"B_MA_SKZ_HydraulikEin"	MB 132	BYTE	// MA: Schrittkette Hydraulik Ein
"B_MA_SKZ_Schmierung"	MB 133	BYTE	// MA: Schrittkette Schmierung
"B_MA_SKZ_Schmierzyklus"	MB 134	BYTE	// MA: Schrittkette Schmierzyklus
"B_MA_Entprell_Zaehler"	MB 135	BYTE	// MA: Entprellzaehler Schmierzyklus
"MB_RDY_M180_189"	MB 144	BYTE	// M180_189: Rückmeldungen
"MB_LED_Zustand_Retten"	MB 151	BYTE
"LED_Zustand_Retten"	MB 154	BYTE	// LED Zustand  retten bei Baustein FC_BHG
"B_MAG_SKZ_Magazin"	MB 162	BYTE	// MAG: Schrittkettenzaehler Magazin
"MB_SKZ_FD_SCHMIERUNG"	MB 163	BYTE
"B_SKZ_Ablauf"	MB 172	BYTE	// WZW: SKZ Ablauf
"B_MAG_SKZ_Unterbrechung"	MB 174	BYTE	// MAG: Schrittkettenzaehler Magunterbrechung
"MB_Zähler_Satus"	MB 177	BYTE	// Zähler im Statusmodul PW
"B_Pos_Speicher"	MB 178	BYTE	// PW: Pos Speicher
"B_Pos_Speicher_Alt"	MB 184	BYTE	// PW: Pos Speicher Alt
"MB_Bruch1"	MB 185	BYTE	// PW: SKZ Fehlermodul
"MB_PW_Pos"	MB 188	BYTE	// SKZ Palettenträger drehen
"MB_WZSP_beide_As_1"	MB 192	BYTE	// WSP: Zaehler f. Verzoeg. beide Eingaenge 1 Signal
"MB_SKZ_PWAblauf"	MB 193	BYTE	// PW: SKZ Ablauf
"MB_WZSP_SKZ_Ablaufmodul"	MB 194	BYTE	// WSP: Schrittkettenzaehler Ablaufmodul Werkzeugspanner
"MB_Counter_Verzoe_Oeffn"	MB 196	BYTE	// WSP: Zaehler fuer verzoegertes oeffnen
"MB_Counter_Verzoe_NotAus"	MB 198	BYTE	// WSP: Zaehler fuer Verzoegerung nach Not-Aus und M6 Request
"MB_INIT_ASUP"	MB 200	BYTE	// ASUP:Initialisierung
"Start_ASUP_Machine"	MB 201	BYTE	// ASUP-fc201
"MB_START_ASUP`S"	MB 202	BYTE
"Start_ASUP_Frame"	MB 203	BYTE	// ASUP-fc203
"MB_A_ASpOV"	MB 204	BYTE
"MB_SKZ_Feierabend"	MB 211	BYTE	// PID: Schrittkettenzähler Feierabendschaltung
"B_SPos_Speicher"	MB 220	BYTE	// SCHWENKKOPF:Pos Speicher
"B_SPos_Speicher_Alt"	MB 221	BYTE	// SCHWENKKOPF:Pos Speicher Alt
"B_SKZ_SErr"	MB 222	BYTE	// SCHWENKKOPF:SKZ Fehlermodul
"B_SKZ_SStat"	MB 223	BYTE	// SCHWENKKOPF:SKZ Statusmodul
"B_SK_Ablauf"	MB 226	BYTE	// SCHWENKKOPF:SKZ Ablauf
"MB_aktiver_Verfahrbereic"	MB 228	BYTE
"MB_SKR_SKZ"	MB 230	BYTE	// SOFTKEYRETTUNG: Schrittkettenzaehler
"M_SPF_SKZ"	MB 242	BYTE	// SPF: Schrittkettenzaehler Spaenefoerderer
"MB_SPF_Zeit_Zaehler"	MB 243	BYTE	// SPF: Zähler für Spänefoerderer Zeiten
"MB_SKZ_RundachsAnf"	MB 247	BYTE	// AX: SKZ Anforderungen Rundachsmodul
"MB_5Achs_Typ"	MB 250	BYTE	// AX: Typ der 5 Achse
"MB_6Achs_Typ"	MB 251	BYTE	// AX: Typ der 10. Achse 6-te Seite
"MB_M10_11_Achse"	MB 256	BYTE	// AX: Zurordnung Achse M10/11
"MB_M22_23_Achse"	MB 257	BYTE	// AX: Zurordnung Achse M22/23
"MB_M32_33_Achse"	MB 258	BYTE	// AX: Zurordnung Achse M32/33
"MB_4Achs_Typ"	MB 259	BYTE	// AX: Typ der 4 Achse
"MB_4Achs_Konfig"	MB 262	BYTE	// AX: Konfiguration der 4. Achse
"MB_5Achs_Konfig"	MB 263	BYTE	// AX: Konfiguration der 5. Achse
"MB_6Achs_Konfig"	MB 264	BYTE	// AX: Konfiguration der 10. Achse 6-te Seite
"MB_SKZ_4ACHS"	MB 265	BYTE	// AX: Schrittkettenzaehler 4. Achse
"MB_SKZ_5ACHS"	MB 266	BYTE	// AX: Schrittkettenzaehler 5./11. Achse
"MB_SKZ_6ACHS"	MB 267	BYTE
"MB_FD_SCHM_HUEBE"	MB 271	BYTE
"MB_FD_ANZAHL_SCHMIERHUB"	MB 272	BYTE
"M_SKZ_Be_Entladen"	MB 292	BYTE	// WZW: SKZ Be-/Entladen
"B_SKZ_Reinig"	MB 294	BYTE	// WZW: Schrittkette Reinigen
"MB_Wiko_NCSNR_alt"	MB 305	BYTE
"B_LS_Pos_Speicher"	MB 311	BYTE
"B_LS_Pos_Speicher_Alt"	MB 312	BYTE
"B_SKZ_LS_Werr"	MB 313	BYTE
"MB_SKZ_Transport"	MB 314	BYTE
"MB_SKZ_Drehstation"	MB 323	BYTE
"MB_SKZ_VERTMAG_WZW"	MB 369	BYTE
"MB_I_DM_ACHSTASTEN"	MB 370	BYTE	// MB-EINGANG: MSST Achstasten 1
"MB_KMTL_DS1_Zahler"	MB 380	BYTE
"MB_KMTL_DS2_Zahler"	MB 381	BYTE
"MB_VS_Korr_BHG"	MB 395	BYTE
"MB_Eil_Korr_BHG"	MB 396	BYTE
"A_Status_FC_PROG_LOAD"	MB 406	BYTE	// A-Status-Meldung von Baustein FC_PROG_LOAD_UNLOAD
"A_Error_FC_PROG_LOAD"	MB 407	BYTE	// A-Error-Meldung von Baustein FC_PROG_LOAD_UNLOAD
"MB_SKZ_Hub_PS"	MB 412	BYTE
"MB_SPF_links_rechts"	MB 429	BYTE
"MB_A_SpOV"	MB 468	BYTE	// Spindeloverride
"MB_SKZ_Getriebe"	MB 469	BYTE	// Getriebe: Schrittkettenzaehler
"MB_Getr_AnzVersuch"	MB 470	BYTE	// Getriebe: Anzahl Versuche
"B_SKZ_SFKSchmieroel"	MB 471	BYTE	// SS: SKZ Schmieröl Spindel
"MB_Werkzeugbruch"	MB 500	BYTE
"MB_WZW_SKZ_Old"	MB 501	BYTE
"MB_AX11_Positionierung"	MB 502	BYTE
"MB_SKZ_NCTAchse"	MB 504	BYTE
"MB_NCTAchs_Typ"	MB 516	BYTE	// AX: Typ der 11. Achse (NC-Teilapperat)
"MB_NCTAchs_Konfig"	MB 517	BYTE	// AX: Konfiguration der 11. Achse (NC-Teilapperat)
"MB_Kegelreinigung_VM_SKZ"	MB 548	BYTE
"mb_hmi_pro_zeilennummer"	MB 554	BYTE	// HMI-PRO: Einrichtzeilennummer
"MB_Palnum_auf_Uebergabep"	MB 556	BYTE	// Palettennummer auf Übergabeplatz
"I_Direkttasten_links"	MB 588	BYTE	// HMI-PRO: OP12/OP15A Direkttasten links
"I_Direkttasten_rechts"	MB 589	BYTE	// HMI-PRO: OP12/OP15A Direkttasten rechts
"MB_ADRESS_BYTE_1_EROWA"	MB 602	BYTE	// Adress Byte 1 der EROWA Schnittstelle
"MB_ADRESS_BYTE_2_EROWA"	MB 603	BYTE	// Adress Byte 2 der EROWA Schnittstelle
"MB_RPC_MODE"	MB 629	BYTE
"MB_RPC_MODE_OLD"	MB 630	BYTE
"MB_ACCESS_LEVEL"	MB 707	BYTE
"IB_GEN_OM_BYTE"	MB 708	BYTE	// Merkereingangsbyte von Smartkey-Reader
"MB_SMARTKEY_BYTE_1"	MB 814	BYTE
"MB_SMARTKEY_AUTHOR"	MB 815	BYTE	// Einstellung des Smartkey Identifizierung
"MB_SF_Rechen1_Co_Vor"	MB 1090	BYTE	// Zähler Sollposition Rechen1 vor  nicht erreicht
"MB_SF_Rechen1_Co_Zurueck"	MB 1091	BYTE	// Zähler Sollposition Rechen1 zurück  nicht erreicht
"MB_SF_Rechen2_Co_Vor"	MB 1095	BYTE
"MB_SF_Rechen2_Co_Zurueck"	MB 1096	BYTE	// Zähler Sollposition Rechen2 zurück  nicht erreicht
"MB_Tisch_Zeit Klem"	MB 1097	BYTE	// Zeit  Druckerhoehung Tisch Achse 200Bar
"MB_Tisch_Takt"	MB 1098	BYTE	// Zähler Tisch geklemmt bei Drucherhoehung 200 Bar
"MB_PERIPHERIE_E_BYTE66"	MB 2066	BYTE	// Zwischenspeicher Peripherie-Eingangsbyte 66
"MB_PERIPHERIE_E_BYTE63"	MB 2067	BYTE	// Zwischenspeicher Peripherie-Eingangsbyte 63
"MB_PERIPHERIE_E_BYTE505"	MB 2068	BYTE	// Digitaleingabemodul , PROFIsafe V2 (PEB505 = DB18.DBB38)
"MB_PERIPHERIE_A_BYTE76"	MB 2076	BYTE	// Zwischenspeicher Peripherie-Ausgangsbyte 76
"MD_VIBS_Eing_SP"	MD 328	REAL	// Skalierte Eingangsspannung des Vibrationssensors
"MD_Restweg_Ax3"	MD 422	REAL
"MD_TDS_FC197"	MD 478	DWORD
"MD_SPI_SPEED_ABS"	MD 726	REAL	// Betragswert der aktuellen Ist-Spindeldrehzahl
"MD_MAPAL_PROFIL"	MD 2040	DWORD	// Angewähltes Profil der U-Achse Mapal
"MW_Wort_0"	MW 0	WORD
"MW_Wort_2"	MW 2	WORD
"MW_Wort_4"	MW 4	WORD
"SpTransp_holen_von"	MW 30	WORD
"SpTransp_bringen_zu"	MW 32	WORD
"MW_BHG_Vorschub"	MW 40	WORD
"MW_DrehDurch_Zaehler"	MW 62	WORD	// DrehDurchführung: Zaehler
"MW_Nr_Bereitst"	MW 64	INT	// WZV: Bereitstellungsplatznummer
"MW_Mag_Plaetze_verfahren"	MW 76	WORD	// GT MAG1: Anzahl verfahrene Paletze bei Ref. Punkt suchen
"MW_Max_ZaehlImpuls"	MW 78	WORD	// GT MAG1: Maximale Zeit Aenderung Zaehlimpuls
"MW_MAG_TMP_Anforderung"	MW 100	WORD	// WZV: T Befehl Platz Anforderung
"MW_MAG_TMMP_Anforderung"	MW 102	WORD	// WZV: TM Platz Anforderung
"MW_Wert_Vibrsensor"	MW 116	INT	// Wert von Vibrationssensor
"I_FD_PT100"	MW 118	WORD	// Temperatursensor Pt100 Fraes-Drehtisch
"W_CHAN1_Flanken"	MW 122	WORD	// Kanal1 Flanken
"MW_Anz_Achs_SA"	MW 128	INT	// Anzahl Achsen Sonderbetriebsart
"MW_MAG_MP_Anforderung"	MW 164	WORD	// MAG: Magazinplatz Anforderung
"MW_MAG_MP_Ist"	MW 166	WORD	// MAG: Magazinplatz Istwert
"MW_MAG_MP_Soll"	MW 168	WORD	// MAG: Magazinplatz Sollwert
"MW_4A_Zust_Stern_Dreieck"	MW 174	WORD
"MW_Zeit_Feierabend"	MW 212	WORD	// PID: Zeitzähler Feierabendschaltung
"MW_BHG"	MW 218	INT
"MW_SFunct1"	MW 274	WORD
"Z_MW_ZYkl_Kratzf."	MW 276	WORD	// KMTL: Zeitzähler Kratzförderer
"MW_Kuehl_Agg_Count"	MW 278	WORD
"MW_SKZ_PWAblauf"	MW 324	INT
"MW_TNUMMER_WZLISTE"	MW 325	INT
"MW_WMR_CNC_EMPF_STORE"	MW 348	INT
"MW_OW_WMR_CNC_SENDEN"	MW 350	WORD	// OW_WMR_CNC_SENDEN vom letzten PLC-Zyklus
"MW_PW_Anwahl_Typ"	MW 362	INT
"MW_PW_Anwahl_Option"	MW 364	INT
"MW_PW_Anwahl_Option2"	MW 366	INT
"O_KM_PROP_VENTIL2"	MW 398	INT	// Proportionalventil Kuehlmittel Hochdruckkreis 80bar
"MW_RET_VAL_SCALE"	MW 402	WORD
"MW_RPL_Bereich"	MW 408	INT
"MW_RPL_Position"	MW 410	INT
"MW_Zaehler_in_Bereich"	MW 415	WORD
"I_HCD1_MAL"	MW 422	INT	// MW-Eingang: Spannhydraulik Druckueberwachung Maschine
"I_HCD1_SST"	MW 424	INT	// MW-Eingang: Spannhydraulik Druckueberwachung Ruestplatz
"MW_SFunct"	MW 464	WORD	// S-Wert
"MW_Zust_Stern_Dreieck"	MW 466	WORD	// Stern Dreieck: Zustandszähler
"MW_SpiSchm_Zaehler"	MW 472	WORD	// Spindel-Schmierung Zähler
"MW_Mess_Nr"	MW 482	INT
"O_BIS_C_35"	MW 484	WORD	// Balluff
"MW_A_Position"	MW 486	WORD
"I_BIS_C_35"	MW 488	WORD	// MW-EINGÄNGE:
"MW_STATE_AXPOSLESEN"	MW 490	WORD
"O_BIS_C_35_1"	MW 492	WORD
"MW_SHOPM_Werkzeugkennung"	MW 494	WORD
"ErrCode_FC_SIEM_PLC_NCK"	MW 496	INT	// ErrCode von Baustein FC_SIEM_PLC_NCK
"WZV_T-Daten"	MW 498	WORD	// WZV: T-Daten neu lesen
"MW_Status_TM_TRANS"	MW 502	WORD
"O_BIS_C_35_2"	MW 504	WORD
"M_WZV_Gr2_WST"	MW 508	WORD	// WZV Zwischenspeicher asynchron Ablegen im Magazin
"MW_ERROR_TM_TRANS"	MW 510	WORD
"I_SPI_TEMP_LAG_HINTEN"	MW 512	WORD	// MW-EINGÄNGE:
"I_Temp_Analog_2"	MW 514	WORD	// MW-EINGÄNGE:
"O_KM_PROP_VENTIL1"	MW 518	INT	// MW-AUSGANG: Kühlmittel Hochdruck PROP-Ventil
"MW_Num_Chanels"	MW 542	WORD
"MW_WFK_NC_SNR"	MW 544	INT
"MW_WK_Nummer"	MW 546	INT
"O_VMS_SPI_SPEED_RPM"	MW 558	WORD
"MW_Greifer_ausfahren_SKZ"	MW 562	INT
"MW_numMagPlaceParam"	MW 570	INT	// Anzahl PArameter Magazinplaetze
"MW_Kegelreinigung_VM_SKZ"	MW 586	INT
"MW_SPF_Zeit_Zaehler"	MW 592	WORD
"MW_WERKSTUECK_ADRESSE"	MW 604	WORD	// Handlingsystem Werkstück Adresse aus H-Fkt 65 bzw. PAR2 in DM_M65
"MW_SERIELLE_ADRESSE"	MW 606	WORD	// Handlingsystem Serielle Adresse Komplett
"MW_ADRESSE_KONTR"	MW 610	WORD
"MW_VMS_SPI_SPEED_RPM"	MW 612	INT	// Analogausgang Vibrationssensor Spindeldrehzahl
"MW_VMS_VIBRATION_SPINDLE"	MW 616	INT	// Analogeingang Vibrationssensor Schwinggeschwindigkeit veff
"MW_RET_VAL_UNSCALE"	MW 618	WORD
"MW_STATUS_MASCH"	MW 624	WORD
"MW_STATUSMASCH_OLD"	MW 626	WORD
"MW_Teilung_RPL"	MW 650	INT
"MW_Teilung_RPL_alt"	MW 652	INT
"I_MACH_BED_T_COMP"	MW 664	WORD
"I_SPI_TEMP_BEA_FRONT"	MW 666	WORD
"I_VMS_VIBRATION_SPINDLE"	MW 668	WORD
"I_TUNING_CPU_KSA_0"	MW 674	WORD
"I_TUNING_CPU_KSA_1"	MW 676	WORD
"I_TUNING_CPU_KSA_2"	MW 678	WORD
"I_TUNING_CPU_KSA_3"	MW 680	WORD
"I_TUNING_CPU_KSA_4"	MW 682	WORD
"O_TUNING_CPU_KSA_0"	MW 684	WORD
"O_TUNING_CPU_KSA_1"	MW 686	WORD
"O_TUNING_CPU_KSA_2"	MW 688	WORD
"O_TUNING_CPU_KSA_3"	MW 690	WORD
"O_TUNING_CPU_KSA_4"	MW 692	WORD
"I_SPI_WZ_SPA"	MW 700	WORD	// Analoger Werkzeugspanner der Spindel
"I_SPI_VERLAG_SENSOR"	MW 702	WORD	// Axiale Wellenverlagerung Startwert Uzo GMN Spindel
"I_ML_SPI_1"	MW 710	WORD	// Merkerwort Eingang  MMS-Vogel
"O_ML_SPI_1"	MW 712	WORD	// Merkerwort Ausgang MMS-Vogel
"MW_SPI_REF_Zeitintervall"	MW 730	WORD	// Spindelüberwachung: Zeitintervall für Spindel Referenzlauf
"MW_PW_TIME_senken"	MW 736	INT	// Time Hub senken  bis PW in Mittelstellung
"MW_PW_Time_ausbl_kon"	MW 738	INT	// Zeitvorgabe Spuel-Konenluftleitung ausblasen
"MW_PW_Time_Spuel_resu"	MW 740	INT	// Resultierende Spuelzeit beim PW senken
"MW_PW_Time_spuel_senk"	MW 742	S5TIME	// Spuelzeit PW-Hub senken ohne Positionsschalter4
"MW_PW_Time_Zeitr_ausbl"	MW 744	S5TIME	// Timer ausblasen Konen
"MW_GetTNR_State"	MW 862	WORD	// State von Call GET_TNR
"MW_Get_Toolstate_State"	MW 864	WORD
"MW1_Get_Toolstate_State"	MW 866	WORD
"I_GEN_POWERMEAS_SPI"	MW 1086	WORD	// MW-Eingänge: Analogeingang Messung Leistung Hauptantrieb
"I_GEN_FLC_COOL_AG_2"	MW 1088	WORD	// MW-Eingänge: Messeinrichtung Kuehlmittel 2
"I_SPI_TEMP_LAG_VORNE"	MW 1092	WORD
"State_FB_SIEM_PUT_GUDs"	MW 1100	WORD	// State-meldung von Baustein FB_SIEM_PUT beim Ablegen der GUDs
"I_SPI_KABEL_PT100_1"	MW 1102	WORD	// MW-EINGÄNGE: Temperatursensor 1 Leitungsueberwachung Hauptantrieb
"I_SPI_KABEL_PT100_2"	MW 1104	WORD	// MW-EINGÄNGE: Temperatursensor 2 Leitungsueberwachung Hauptantrieb
"I_SPI_TEMP"	MW 1106	WORD
"I_MASCH_BETT_T_KOMP"	MW 1120	WORD	// MW-EINGÄNGE: Temperatursensor Maschinenbett PT 100
"I_SPI_PT100"	MW 1122	WORD	// MW-EINGÄNGE: Lager-Temperatursensor PT100 Hauptantrieb
"I_VSP_TEMP"	MW 1124	WORD
"I_SPI_TEMP_MONITOR"	MW 2000	WORD	// MW-EINGÄNGE: Temperaturüberwachung Spindelstock (55/65H)
"I_RESERVE_4_33"	MW 2002	WORD	// MW-EINGÄNGE: Dummy für Hardware 55H
"OB_ZYKLISCH"	OB 1	OB 1	// Zyklische Programmbearbeitung
"TOD_INT0"	OB 10	OB 10	// Time of Day Interrupt 0
"OB_WECKALARM1"	OB 35	OB 35	// Cyclic Interrupt 1
"OB_PROZESSALARM1"	OB 40	OB 40	// Prozessalarm 1
"OB_I_O_FLT1"	OB 82	OB 82	// I/O Point Fault 1
"OB_PRG_ABL_FEHLER"	OB 85	OB 85	// OB Programmablauffehler
"OB_RACK_FLT"	OB 86	OB 86	// Loss of Rack Fault
"OB_WARMSTART1"	OB 100	OB 100	// Hochlauf / Neustart
"OB_PROG_ERR"	OB 121	OB 121	// Programming Error
"OB_MOD_ERR"	OB 122	OB 122	// Module Access Error
"IB_HCD_AV_CL_PO_1_SST_H"	PIB 430	BYTE
"IB_HCD_AV_CL_PO_1_SST_L"	PIB 431	BYTE
"IB_HCD_AV_CL_PO_2_SST_H"	PIB 432	BYTE
"IB_HCD_AV_CL_PO_2_SST_L"	PIB 433	BYTE
"IB_HCD_AV_CL_PO_3_SST_H"	PIB 434	BYTE
"IB_HCD_AV_CL_PO_3_SST_L"	PIB 435	BYTE
"IB_HCD_AV_CL_PO_4_SST_H"	PIB 436	BYTE
"IB_HCD_AV_CL_PO_4_SST_L"	PIB 437	BYTE
"IB_HCD_AV_CL_PO_1_MPL_H"	PIB 438	BYTE
"IB_HCD_AV_CL_PO_1_MPL_L"	PIB 439	BYTE
"IB_HCD_AV_CL_PO_2_MPL_H"	PIB 440	BYTE
"IB_HCD_AV_CL_PO_2_MPL_L"	PIB 441	BYTE
"IB_HCD_AV_CL_PO_3_MPL_H"	PIB 442	BYTE
"IB_HCD_AV_CL_PO_3_MPL_L"	PIB 443	BYTE
"IB_HCD_AV_CL_PO_4_MPL_H"	PIB 444	BYTE
"IB_HCD_AV_CL_PO_4_MPL_L"	PIB 445	BYTE
"IB_HCD_STATE_CL_PO_1_SST"	PIB 446	BYTE
"IB_HCD_STATE_CL_PO_2_SST"	PIB 447	BYTE
"IB_HCD_STATE_CL_PO_3_SST"	PIB 448	BYTE
"IB_HCD_STATE_CL_PO_4_SST"	PIB 449	BYTE
"IB_HCD_STATE_CL_PO_1_MPL"	PIB 450	BYTE
"IB_HCD_STATE_CL_PO_2_MPL"	PIB 451	BYTE
"IB_HCD_STATE_CL_PO_3_MPL"	PIB 452	BYTE
"IB_HCD_STATE_CL_PO_4_MPL"	PIB 453	BYTE
"IB_HCD_DIAG_SOFTWARE"	PIB 454	BYTE
"IB_HCD_DIAG_MPL_SST"	PIB 455	BYTE
"IB_HCD_MI_TURNT_INP"	PIB 456	BYTE
"IB_SP_P_IST_ST_1_RPL_H"	PIB 1000	BYTE	// HAWE-Box:
"IB_SP_P_IST_ST_1_RPL_L"	PIB 1001	BYTE	// HAWE-Box:
"IB_SP_P_IST_ST_2_RPL_H"	PIB 1002	BYTE	// HAWE-Box:
"IB_SP_P_IST_ST_2_RPL_L"	PIB 1003	BYTE	// HAWE-Box:
"IB_SP_P_IST_ST_3_RPL_H"	PIB 1004	BYTE	// HAWE-Box:
"IB_SP_P_IST_ST_3_RPL_L"	PIB 1005	BYTE	// HAWE-Box:
"IB_SP_P_IST_ST_4_RPL_H"	PIB 1006	BYTE	// HAWE-Box:
"IB_SP_P_IST_ST_4_RPL_L"	PIB 1007	BYTE	// HAWE-Box:
"IB_SP_P_IST_ST_1_MPL_H"	PIB 1008	BYTE	// HAWE-Box:
"IB_SP_P_IST_ST_1_MPL_L"	PIB 1009	BYTE	// HAWE-Box:
"IB_SP_P_IST_ST_2_MPL_H"	PIB 1010	BYTE	// HAWE-Box:
"IB_SP_P_IST_ST_2_MPL_L"	PIB 1011	BYTE	// HAWE-Box:
"IB_SP_P_IST_ST_3_MPL_H"	PIB 1012	BYTE	// HAWE-Box:
"IB_SP_P_IST_ST_3_MPL_L"	PIB 1013	BYTE	// HAWE-Box:
"IB_SP_P_IST_ST_4_MPL_H"	PIB 1014	BYTE	// HAWE-Box:
"IB_SP_P_IST_ST_4_MPL_L"	PIB 1015	BYTE	// HAWE-Box:
"IB_SP_STATE_ST_1_RPL"	PIB 1016	BYTE	// HAWE-Box:
"IB_SP_STATE_ST_2_RPL"	PIB 1017	BYTE	// HAWE-Box:
"IB_SP_STATE_ST_3_RPL"	PIB 1018	BYTE	// HAWE-Box:
"IB_SP_STATE_ST_4_RPL"	PIB 1019	BYTE	// HAWE-Box:
"IB_SP_STATE_ST_1_MPL"	PIB 1020	BYTE	// HAWE-Box:
"IB_SP_STATE_ST_2_MPL"	PIB 1021	BYTE	// HAWE-Box:
"IB_SP_STATE_ST_3_MPL"	PIB 1022	BYTE	// HAWE-Box:
"IB_SP_STATE_ST_4_MPL"	PIB 1023	BYTE	// HAWE-Box:
"IB_SP_FUNKTION_MPL_RPL"	PIB 1024	BYTE	// HAWE-Box:
"IB_SP_DIAGNOSE_MPL_RPL"	PIB 1025	BYTE	// HAWE-Box:
"IB_TOOL_CUT_FORCE_1_MON"	PIB 1300	BYTE	// ARTIS/Toolinspect Eingangs-Byte 1
"IW_Tuning_CPU_0"	PIW 210	WORD	// xx-xx.x ME Datenschnittstelle Profibus(8)
"IW_Tuning_CPU_1"	PIW 212	WORD	// xx-xx.x ME Datenschnittstelle Profibus(8)
"IW_Tuning_CPU_2"	PIW 214	WORD	// xx-xx.x ME Datenschnittstelle Profibus(8)
"IW_Tuning_CPU_3"	PIW 216	WORD	// xx-xx.x ME Datenschnittstelle Profibus(8)
"IW_Tuning_CPU_4"	PIW 218	WORD	// xx-xx.x ME Datenschnittstelle Profibus(8)
"IW_TUNING_CPU_5"	PIW 220	WORD	// xx-xx.x ME Datenschnittstelle Profibus(8)
"IW_WMR_CNC_0"	PIW 258	WORD	// REGAL EXTERN Bit-Orientiertes Eingangswort 0
"IW_WMR_CNC_1"	PIW 260	WORD	// REGAL EXTERN Bit-Orientiertes Eingangswort 1
"IW_WMR_CNC_MAINCOMMAND"	PIW 262	WORD	// REGAL EXTERN Hauptkommando Nutzdaten
"IW_WMR_CNC_SUBCOMMAND"	PIW 264	WORD	// REGAL EXTERN Unterkommando Nutzdaten
"IW_WMR_CNC_1_DATA"	PIW 266	WORD	// REGAL EXTERN Kennung Nutzdaten 1 Wort
"IW_WMR_CNC_2_DATA"	PIW 268	WORD	// REGAL EXTERN Kennung Nutzdaten 2 Wort
"IW_WMR_CNC_SENDEN"	PIW 270	WORD	// REGAL EXTERN Handshake senden Zaehler
"IW_WMR_CNC_EMPFANGEN"	PIW 272	WORD	// REGAL EXTERN Handshake empfangen Zaehler
"IW_TUNING_CPU_CU_0"	PIW 300	WORD
"IW_TUNING_CPU_CU_1"	PIW 302	WORD
"IW_TUNING_CPU_CU_2"	PIW 304	WORD
"IW_TUNING_CPU_CU_3"	PIW 306	WORD
"IW_TUNING_CPU_CU_4"	PIW 308	WORD
"IW_SP_Wort_24"	PIW 334	WORD	// SpannHydraulik Wort 24
"IW_BIS_C_35"	PIW 1060	WORD
"IW_ROBOT_0"	PIW 1160	WORD	// xx-xx.x ME Start-Adr: Roboter-Schnittstelle - DPDP-Koppler
"OB_HCD_SV_CL_PO_1_SST_H"	PQB 430	BYTE
"OB_HCD_SV_CL_PO_1_SST_L"	PQB 431	BYTE
"OB_HCD_SV_CL_PO_2_SST_H"	PQB 432	BYTE
"OB_HCD_SV_CL_PO_2_SST_L"	PQB 433	BYTE
"OB_HCD_SV_CL_PO_3_SST_H"	PQB 434	BYTE
"OB_HCD_SV_CL_PO_3_SST_L"	PQB 435	BYTE
"OB_HCD_SV_CL_PO_4_SST_H"	PQB 436	BYTE
"OB_HCD_SV_CL_PO_4_SST_L"	PQB 437	BYTE
"OB_HCD_SV_CL_PO_1_MPL_H"	PQB 438	BYTE
"OB_HCD_SV_CL_PO_1_MPL_L"	PQB 439	BYTE
"OB_HCD_SV_CL_PO_2_MPL_H"	PQB 440	BYTE
"OB_HCD_SV_CL_PO_2_MPL_L"	PQB 441	BYTE
"OB_HCD_SV_CL_PO_3_MPL_H"	PQB 442	BYTE
"OB_HCD_SV_CL_PO_3_MPL_L"	PQB 443	BYTE
"OB_HCD_SV_CL_PO_4_MPL_H"	PQB 444	BYTE
"OB_HCD_SV_CL_PO_4_MPL_L"	PQB 445	BYTE
"OB_HCD_STATE_CL_PO_1_SST"	PQB 446	BYTE
"OB_HCD_STATE_CL_PO_2_SST"	PQB 447	BYTE
"OB_HCD_STATE_CL_PO_3_SST"	PQB 448	BYTE
"OB_HCD_STATE_CL_PO_4_SST"	PQB 449	BYTE
"OB_HCD_STATE_CL_PO_1_MPL"	PQB 450	BYTE
"OB_HCD_STATE_CL_PO_2_MPL"	PQB 451	BYTE
"OB_HCD_STATE_CL_PO_3_MPL"	PQB 452	BYTE
"OB_HCD_STATE_CL_PO_4_MPL"	PQB 453	BYTE
"OB_HCD_FCT_MPL_SST"	PQB 454	BYTE
"OB_HCD_DIAG_MPL_SST"	PQB 455	BYTE
"OB_HCD_TOL_VAL_PRE_REA"	PQB 456	BYTE
"OB_HCD_TOL_VAL_READJUST"	PQB 457	BYTE
"OB_HCD_TOL_VAL_EMSTP"	PQB 458	BYTE
"OB_HCD_DELTA_CONTROL"	PQB 459	BYTE
"OB_HCD_DELTA_REGULATION"	PQB 460	BYTE
"OB_HCD_PRESSURE_RELEASE"	PQB 461	BYTE
"OB_HCD_PRE_RET_VALV_OPEN"	PQB 462	BYTE
"OB_HCD_TIME_DELAY_CLAMP"	PQB 463	BYTE
"OB_HCD_RT_RET_VAL_OPEN"	PQB 464	BYTE
"OB_SP_P_SOLL_ST_1_RPL_H"	PQB 1000	BYTE	// HAWE-Box:
"OB_SP_P_SOLL_ST_1_RPL_L"	PQB 1001	BYTE	// HAWE-Box:
"OB_SP_P_SOLL_ST_2_RPL_H"	PQB 1002	BYTE	// HAWE-Box:
"OB_SP_P_SOLL_ST_2_RPL_L"	PQB 1003	BYTE	// HAWE-Box:
"OB_SP_P_SOLL_ST_3_RPL_H"	PQB 1004	BYTE	// HAWE-Box:
"OB_SP_P_SOLL_ST_3_RPL_L"	PQB 1005	BYTE	// HAWE-Box:
"OB_SP_P_SOLL_ST_4_RPL_H"	PQB 1006	BYTE	// HAWE-Box:
"OB_SP_P_SOLL_ST_4_RPL_L"	PQB 1007	BYTE	// HAWE-Box:
"OB_SP_P_SOLL_ST_1_MPL_H"	PQB 1008	BYTE	// HAWE-Box:
"OB_SP_P_SOLL_ST_1_MPL_L"	PQB 1009	BYTE	// HAWE-Box:
"OB_SP_P_SOLL_ST_2_MPL_H"	PQB 1010	BYTE	// HAWE-Box:
"OB_SP_P_SOLL_ST_2_MPL_L"	PQB 1011	BYTE	// HAWE-Box:
"OB_SP_P_SOLL_ST_3_MPL_H"	PQB 1012	BYTE	// HAWE-Box:
"OB_SP_P_SOLL_ST_3_MPL_L"	PQB 1013	BYTE	// HAWE-Box:
"OB_SP_P_SOLL_ST_4_MPL_H"	PQB 1014	BYTE	// HAWE-Box:
"OB_SP_P_SOLL_ST_4_MPL_L"	PQB 1015	BYTE	// HAWE-Box:
"OB_SP_STATE_ST_1_RPL"	PQB 1016	BYTE	// HAWE-Box:
"OB_SP_STATE_ST_2_RPL"	PQB 1017	BYTE	// HAWE-Box:
"OB_SP_STATE_ST_3_RPL"	PQB 1018	BYTE	// HAWE-Box:
"OB_SP_STATE_ST_4_RPL"	PQB 1019	BYTE	// HAWE-Box:
"OB_SP_STATE_ST_1_MPL"	PQB 1020	BYTE	// HAWE-Box:
"OB_SP_STATE_ST_2_MPL"	PQB 1021	BYTE	// HAWE-Box:
"OB_SP_STATE_ST_3_MPL"	PQB 1022	BYTE	// HAWE-Box:
"OB_SP_STATE_ST_4_MPL"	PQB 1023	BYTE	// HAWE-Box:
"OB_SP_FUNKTION_MPL_RPL"	PQB 1024	BYTE	// HAWE-Box:
"OB_SP_DIAGNOSE_MPL_RPL"	PQB 1025	BYTE	// HAWE-Box:
"OB_SP_P_TOL_DRUCK_ERREIC"	PQB 1026	BYTE	// HAWE-Box:
"OB_SP_P_TOL_NACHREGELN"	PQB 1027	BYTE	// HAWE-Box:
"OB_SP_P_TOL_NOTAUS"	PQB 1028	BYTE	// HAWE-Box:
"OB_SP_DELTA_STEUERUNG"	PQB 1029	BYTE	// HAWE-Box:
"OB_SP_DELTA_REGELUNG"	PQB 1030	BYTE	// HAWE-Box:
"OB_SP_P_LOESEDRUCK"	PQB 1031	BYTE	// HAWE-Box:
"OB_SP_P_DRUCK_RV_OEFFNEN"	PQB 1032	BYTE	// HAWE-Box:
"OB_SP_T_VERZ_SPANNEN"	PQB 1033	BYTE	// HAWE-Box:
"OB_SP_T_RV_OEFFNEN"	PQB 1034	BYTE	// HAWE-Box:
"OB_TOOL_CUT_FORCE_1_MON"	PQB 1300	BYTE	// ARTIS/Toolinspect Ausgangs-Byte 1
"OB_TOOL_CUT_FORCE_2_MON"	PQB 1301	BYTE	// ARTIS/Toolinspect Ausgangs-Byte 2
"OW_Tuning_CPU_0"	PQW 210	WORD	// xx-xx.x MA Datenschnittstelle Profibus(8)
"OW_Tuning_CPU_1"	PQW 212	WORD	// xx-xx.x MA Datenschnittstelle Profibus(8)
"OW_Tuning_CPU_2"	PQW 214	WORD	// xx-xx.x MA Datenschnittstelle Profibus(8)
"OW_Tuning_CPU_3"	PQW 216	WORD	// xx-xx.x MA Datenschnittstelle Profibus(8)
"OW_Tuning_CPU_4"	PQW 218	WORD	// xx-xx.x MA Datenschnittstelle Profibus(8)
"OW_Tuning_CPU_C0"	PQW 220	WORD	// xx-xx.x MA Datenschnittstelle Profibus(8)
"OW_Tuning_CPU_C1"	PQW 222	WORD	// xx-xx.x MA Datenschnittstelle Profibus(8)
"OW_Tuning_CPU_C2"	PQW 224	WORD	// xx-xx.x MA Datenschnittstelle Profibus(8)
"OW_Tuning_CPU_C3"	PQW 226	WORD	// xx-xx.x MA Datenschnittstelle Profibus(8)
"OW_Tuning_CPU_5"	PQW 228	WORD	// xx-xx.x MA Datenschnittstelle Profibus(8)
"OW_Tuning_CPU_6"	PQW 230	WORD	// xx-xx.x MA Datenschnittstelle Profibus(8)
"OW_TUNING_CPU_7"	PQW 232	WORD	// xx-xx.x MA Datenschnittstelle Profibus(8)
"OW_TUNING_CPU_8"	PQW 234	WORD
"OW_WMR_CNC_0"	PQW 258	WORD	// REGAL EXTERN Bit-Orientiertes Ausgangswort 0
"OW_WMR_CNC_1"	PQW 260	WORD	// REGAL EXTERN Bit-Orientiertes Ausgangswort 1
"OW_WMR_CNC_MAINCOMMAND"	PQW 262	WORD	// REGAL EXTERN Hauptkommando Nutzdaten
"OW_WMR_CNC_SUBCOMMAND"	PQW 264	WORD	// REGAL EXTERN Unterkommando Nutzdaten
"OW_WMR_CNC_1_DATA"	PQW 266	WORD	// REGAL EXTERN Kennung Nutzdaten 1 Wort
"OW_WMR_CNC_2_DATA"	PQW 268	WORD	// REGAL EXTERN Kennung Nutzdaten 2 Wort
"OW_WMR_CNC_SENDEN"	PQW 270	WORD	// REGAL EXTERN Handshake senden Zaehler
"OW_WMR_CNC_EMPFANGEN"	PQW 272	WORD	// REGAL EXTERN Handshake empfangen Zaehler
"OW_TUNING_CPU_CU_0"	PQW 300	WORD
"OW_TUNING_CPU_CU_1"	PQW 302	WORD
"OW_TUNING_CPU_CU_2"	PQW 304	WORD
"OW_TUNING_CPU_CU_3"	PQW 306	WORD
"OW_TUNING_CPU_CU_4"	PQW 308	WORD
"OW_TUNING_CPU_CU_5"	PQW 310	WORD
"OW_BIS_C_35"	PQW 1060	WORD	// Balluff
"OW_BIS_C_35_1"	PQW 1062	WORD
"OW_BIS_C_35_2"	PQW 1064	WORD
"OW_ROBOT_0"	PQW 1160	WORD	// xx-xx.x MA Start-Adr: Roboter-Schnittstelle - DPDP-Koppler
"MSSTLED BA AUTO"	Q 0.0	BOOL	// MSST: LED Betriebsart AUTO_LED 21
"DM_LED Spindel links"	Q 0.4	BOOL	// MSST: LED Spindel links_LED 10
"DM_LED Spindel Halt *"	Q 0.5	BOOL	// MSST: LED Spindel Halt *_LED 9
"DM_LED Spindel rechts"	Q 0.6	BOOL	// MSST: LED Spindel rechts_LED 8
"DM_LED Y-Achse plus"	Q 1.4	BOOL	// MSST: LED Y-Achse minus_LED 20
"DM_LED Z-Achse plus(3)"	Q 1.5	BOOL	// MSST: LED Z-Achse plus LED 19
"DM_LED 4-Achse rechts"	Q 1.6	BOOL	// MSST: LED 4-Achse (4)_rechts LED 38
"MSSTLED 1 INC"	Q 2.0	BOOL	// MSST: LED 1 INC_LED 14
"MSSTLED 10 INC"	Q 2.1	BOOL	// MSST: LED 10 INC_LED 24
"MSSTLED 100 INC"	Q 2.2	BOOL	// MSST: LED 100 INC_LED 34
"MSSTLED 1000 INC"	Q 2.3	BOOL	// MSST: LED 1000 INC_LED 44
"MSSTLED var. INC"	Q 2.5	BOOL	// MSST: LED var. INC_LED 4
"DM_LED 5/6Achsanwahl"	Q 4.5	BOOL	// MSST: LED Anwahl 5/6Achse
"DM_LED 5/6-Achse minus"	Q 4.6	BOOL	// MSST: LED 5/6-Achse minus LED 48
"DM_LED 5/6-Achse plus"	Q 4.7	BOOL	// MSST: LED 5/6-Achse plus LED 48
"DM_LED X-Achse minus(1)"	Q 5.0	BOOL	// MSST: LED X-Achse (1) minus LED 28
"DM_LED Eilgang"	Q 5.1	BOOL	// MSST: LED_Eilgang LED 29
"DM_LED X-Achse plus(1)"	Q 5.2	BOOL	// MSST: LED X-Achse (1) plus LED 30
"DM_LED Y-Achse minus"	Q 5.3	BOOL	// MSST: LED Y-Achse plus_LED 38
"DM_LED Z-Achse minus(3)"	Q 5.4	BOOL	// MSST: LED Z. Achse (3)minus_LED 39
"MSSTLED C-Achse (6)"	Q 5.5	BOOL	// MSST: LED C-Achse (6)_LED 40
"DM_LED_MKS_WKS"	Q 6.1	BOOL	// MSST: LED MKS_WKS
"DM_LED SpiOver_erhoeh"	Q 6.4	BOOL	// MSST: LED Spinbdeloverride erhoehen
"DM_LED_SpiOver_100%"	Q 6.5	BOOL	// MSST: LED Spindeloverride 100%
"DM_LED_SpiOver_reduz"	Q 6.6	BOOL	// MSST: LED Spindeloverride reduzieren
"DM_LED IKZ_ein_aus"	Q 7.0	BOOL	// MSST: LED IKZ EIN/AUS
"DM_LED Kühlmittel"	Q 7.1	BOOL	// MSST: LED Kühlmittel EIN/AUS
"DM_LED_WZSpanner"	Q 7.4	BOOL	// MSST: LED Werkzeugspanner auf zu
"OX_AL_XACHS_Bremse_auf"	Q 32.0	BOOL	// Ansteuerung Motorbremse X-Achse
"OX_AL_YACHS_Bremse_auf"	Q 32.1	BOOL	// Ansteuerung Motorbremse Y-Achse
"OX_AL_ZACHS_Bremse_auf"	Q 33.0	BOOL	// Ansteuerung Motorbremse Z-Achse
"OX_AL_4ACHS_Bremse_auf"	Q 33.1	BOOL	// Ansteuerung Motorbremse 4-Achse
"OX_AL_5ACHS_Bremse_auf"	Q 34.0	BOOL	// Ansteuerung Motorbremse 5-Achse
"OX_PW_ACHS_Bremse_auf"	Q 34.1	BOOL	// Achse 8 (PW)  Bremse lüften
"OX_SPI_WYE"	Q 35.0	BOOL	// Stern Dreieck: Ausgang Stern
"OX_SPI_DELTA"	Q 35.1	BOOL	// Stern Dreieck: Ausgang Dreieck
"OX_GEN_PLC_RDY"	Q 36.0	BOOL	// Maschine 'Ein'  (CNC PLC Betriebsbereit)
"OX_WM_Freigabe_re_li"	Q 36.1	BOOL	// Freigabe Werkzeugmagazin
"OX_PC_DOOR_UNLOCK"	Q 36.2	BOOL	// Magnetverriegelung Ruestplatz Palettenwechsler entriegeln
"OX_OMS_ON"	Q 36.3	BOOL	// Nebel- u.Rauchabscheider 'Ein'
"OX_PC_MPL_PALLET_RELEASE"	Q 37.0	BOOL	// Palette auf Tisch lösen
"OX_PC_MPL_PALLET_CLAMP"	Q 37.1	BOOL	// Palette auf Tisch spannen
"OX_SH_CLAMP_CLAMP"	Q 37.2	BOOL	// Schwenkfraeskopf Klemmung klemmen
"OX_SH_CLAMP_RELEASE"	Q 37.3	BOOL	// Schwenkfraeskopf Klemmung loesen
"OX_GEN_AXIS4_CLAMP"	Q 38.0	BOOL	// 4.Achse klemmen
"OX_GEN_AXIS5_CLAMP"	Q 38.1	BOOL	// 5.Achse klemmen
"OX_SPI_LUB_OIL_PUMP_ON"	Q 38.2	BOOL	// Schmierung Hauptantrieb 24.000 U/min
"OX_SPI_LUB_CAIR_ON"	Q 38.3	BOOL	// Schwenkfräskopf Druckluft Schmierung 'Ein'
"OX_GEN_CAIR_ON"	Q 39.0	BOOL	// Pneumatik 'Ein'
"OX_AL_Manual_Betrieb"	Q 39.1	BOOL	// Handbetrieb (Manual)
"OX_HW_CNC_ACTIVE"	Q 39.2	BOOL	// Handkommandostation angewählt /Umschaltung Zustimmtaster
"OX_AL_Start_Sig_Renishaw"	Q 39.3	BOOL	// Messtasterfreigabe
"OX_CC_CU_PUMP"	Q 40.0	BOOL	// Foerderpumpe Kuehlmittel ein
"OX_SPI_TL_CLAMP_RELEASE"	Q 40.1	BOOL	// Werkzeugspanner loesen
"OX_GEN_CABIN_UNLOCK"	Q 40.2	BOOL	// Magnetverriegelung Kabinentüre entriegeln
"OX_TC_CLEAN_EXTEND"	Q 40.3	BOOL	// Werkzeugreinigung zur Stellung Reinigen
"OX_GEN_OM_4_ENABLE"	Q 41.0	BOOL	// Energiefreigabe 4.Betriebsart
"OX_TLB_ENABLE"	Q 41.1	BOOL	// WZB Messung Start
"OX_GEN_HYD_ON"	Q 41.2	BOOL	// Hydraulik 'Ein'
"OX_GEN_CNC_PGM_ACTIVE"	Q 41.3	BOOL	// Betriebsstundenzaehler Programm laeuft
"OX_SH_GEAR_STAGE1"	Q 42.2	BOOL	// Drehzahlschaltung Hauptantrieb mit Getriebe    Drehzahl kle
"OX_SH_GEAR_STAGE2"	Q 42.3	BOOL	// Drehzahlschaltung Hauptantrieb mit Getriebe    Drehzahl gr
"OX_WM_Beladung_entr_auf"	Q 43.0	BOOL	// Freigabe Magnetverriegelung Fenster Werkzeugbestückung (Lampe)
"OX_SPI_CAIR_JETS_EXT"	Q 43.1	BOOL	// Blasluft Kuehlung Werkzeug 'Ein'
"OX_SPI_CAIR_TOOL"	Q 43.2	BOOL	// Druckluft Werkzeugkegel ausblasen
"OX_TC_CLEAN_HOME_POS"	Q 43.3	BOOL	// Werkzeugreinigung zur Grundstellung
"OX_WM_XACHS_Bremse_auf"	Q 44.0	BOOL	// Werkzeugmagazin X-Achse Bremse auf
"OX_LA_CAIR_CLEAN"	Q 44.1	BOOL	// Laser abblasen
"OX_GEN_LUB_ON"	Q 45.0	BOOL	// Schmierung Maschine 'Ein'
"OX_SPI_ROTRA_LUB_ON"	Q 45.1	BOOL	// Dreh-Duchführung Ansteuerung Schmierpumpe 'Ein'
"OX_TC_GRP_FAST_ROTATE"	Q 46.0	BOOL	// Werkstueckgreifer drehen schnell
"OX_TC_GRP_SLOW_ROTATE"	Q 46.1	BOOL	// Werkstueckgreifer drehen langsam
"OX_TC_GRP_1_TOOL_MAG"	Q 46.2	BOOL	// Werkzeuggreifer drehen Richtung Werkzeugmagazin
"OX_TC_GRP_1_SPINDLE"	Q 46.3	BOOL	// Werkzeuggreifer drehen Richtung Spindel
"OX_TC_DOOR_OPEN"	Q 47.0	BOOL	// Werkzeugwechsler Tuer oeffnen
"OX_TC_DOOR_CLOSE"	Q 47.1	BOOL	// Werkzeugwechsler Tuer schliessen
"OX_TC_CYL_1_SPINDLE"	Q 47.2	BOOL	// Werkzeugmagazin Zylinder1 Richtung Spindel
"OX_TC_CYL_1_HOME_POS"	Q 47.3	BOOL	// Werkzeugmagazin Zylinder1 Richtung Grundstellung
"OX_PC_CLAMP_CONE_BL_O"	Q 47.4	BOOL	// Palettenträger Spannstelle ausblasen
"OX_PC_LIFT_FAST_DOWN"	Q 47.5	BOOL	// Hubeinheit Palettenwechsler schnell nach unten
"OX_PC_LIFT_FAST_UP"	Q 47.6	BOOL	// Hubeinheit Palettenwechsler schnell nach oben
"OX_CC_FORWARD"	Q 48.0	BOOL	// Rechtslauf Spaenefoerderer
"OX_CC_BACKWARD"	Q 48.1	BOOL	// Linkslauf Spaenefoerderer
"OX_CC_WORM_ON"	Q 48.2	BOOL	// Spaenefoerderer Schneckenantrieb ein
"OX_CC_WORM_2_ON"	Q 48.3	BOOL	// Spaenefoerderer Schneckenantrieb 2 ein
"OX_MI_TURNT_OPER_HOUR"	Q 48.4	BOOL	// Fraes-Drehtisch Betriebsstundenzaehler
"OX_TC_RETENTION_EXTEND"	Q 49.0	BOOL	// Werkzeug-Rueckhalt ausfahren (verriegeln)
"OX_PW_Ventil_Abfrage"	Q 49.1	BOOL	// Ventil Luftstrom Palette
"OX_WW_GRF_ENTRIEGELN"	Q 49.2	BOOL	// Verriegelung Werkzeuggreifer entriegeln
"OX_ENERGYSAFE"	Q 49.3	BOOL	// Energysafe (Alle Achsen stehen)
"OX_LA_MOVE_OUT"	Q 50.0	BOOL	// Laser: Laser ausfahren
"OX_LA_MOVE_IN"	Q 50.1	BOOL	// Laser: Laser einfahren
"OX_LA_BARR_AIR_OFF"	Q 50.2	BOOL	// Laser: Ventil Sperrluft
"OX_LA_DIRT_TRAP_OPEN"	Q 50.3	BOOL	// Laser: Ventil Schmutzblende
"OX_AL_Messdose_abblasen"	Q 51.0	BOOL	// Blasluft Reinigung Werkzeugvermessung
"OX_LA_TRANSMITTER_ON"	Q 51.1	BOOL	// Laser: Sender Ein
"OX_LA_RECEIVER_ON"	Q 51.2	BOOL	// Laser: Freigabe Laser Empfangsdaten
"OX_LA_RECEIVER_2_ENABLE"	Q 51.3	BOOL	// Laser: Freigabe Laser einschalten 2
"OX_PC_LIFT_UP"	Q 52.0	BOOL	// Palettenwechsler nach oben
"OX_PC_LIFT_DOWN"	Q 52.1	BOOL	// Palettenwechsler nach unten
"OX_PW_0_Grad_Drehen"	Q 52.2	BOOL	// Palettenwechsler schwenken 0 Grad Position
"OX_PW_180_Grad_Drehen"	Q 52.3	BOOL	// Palettenwechsler schwenken 180 Grad Position
"OX_TOOL_MQL_M7"	Q 53.0	BOOL	// Umschaltung Ventil Schmiersystem innere Kuehlmittelzufuhr
"OX_TOOL_MQL_M8"	Q 53.1	BOOL	// Umschaltung Ventil Schmiersystem Kuehlmittel 1
"OX_TOOL_MQL_VAL_1"	Q 53.2	BOOL	// Minimalmengen Schmierung Ventil 1 Ein
"OX_TOOL_MQL_VAL_2"	Q 53.3	BOOL	// Minimalmengen Schmierung Ventil 2 Ein
"OX_CU_M8"	Q 54.0	BOOL	// Pumpe Kühlmittel 1 'Ein' (M8)
"OX_CU_FLUSH_CABIN"	Q 54.1	BOOL	// Spaenespuelung 'Ein'
"OX_CU_PAPER_MOVE"	Q 54.2	BOOL	// Motor Ein Papierbandfilter
"OX_CU_FLUSH_PISTOL"	Q 54.3	BOOL	// Pumpe Kühlmittel Spülpistole
"OX_SPI_RELEASE"	Q 55.0	BOOL	// Fraesspindel loesen
"OX_SPI_CLAMP"	Q 55.1	BOOL	// Fraesspindel klemmen
"OX_MI_TURNT_TAB_CLAMP"	Q 55.2	BOOL	// Klemmung Fraes-Drehtisch klemmen
"OX_MI_TURNT_TAB_RELEASE"	Q 55.3	BOOL	// Klemmung Fraes-Drehtisch loesen
"OX_CU_M7"	Q 56.0	BOOL	// Hochdruckpumpe Kuehlmittel 2.1
"OX_CU_FLUSH_ROOF"	Q 56.1	BOOL	// Pumpe Spaenespuelung Dach
"OX_CU_SUP_F_REG_PUMP_ON"	Q 56.2	BOOL	// Foerderpumpe Feinstbereich
"OX_KM_PUMPE_FILTER_FEINB"	Q 56.3	BOOL	// Foerderpumpe Feinstbereich
"OX_CU_M7_PRESSURE2_ON"	Q 56.6	BOOL	// Kühlmittelanlage Druck2 M7 ein
"OX_CU_M7_PRESSURE1_ON"	Q 56.7	BOOL
"OX_PC_TABLE_FLUSH"	Q 57.0	BOOL	// Ventil Spänespülung Palettenwechsler
"OX_CU_M7_STAGE_2"	Q 57.1	BOOL	// Hochdruckpumpe Kuehlmittel 2 80 bar
"OX_AL_5ACHS_KLE_LOESEN"	Q 57.2	BOOL	// Klemmung loesen NC-Teilapparat
"OX_HCD_SST_LOCK"	Q 57.3	BOOL	// Spannhydraulik Ruestplatz gespannt
"OX_CU_FLUSH_PUMP_PC"	Q 57.4	BOOL	// Pumpe Spänespülung Palettenwechsler
"OX_GEN_SIGNALLAMP_RD"	Q 60.0	BOOL	// Signalleuchte Farbe RD
"OX_GEN_SIGNALLAMP_YE"	Q 60.1	BOOL	// Signalleuchte Farbe YE
"OX_GEN_SIGNALLAMP_GN"	Q 60.2	BOOL	// Signalleuchte Farbe GN
"OX_GEN_SIGNALLAMP_BU"	Q 60.3	BOOL	// Signalleuchte Farbe BU
"OX_PC_PAL_CAR_DOWN"	Q 60.4	BOOL	// Takttisch Palettenträger senken
"OX_PC_PAL_CAR_UP"	Q 60.5	BOOL	// Takttisch Palettenträger heben
"OX_GEN_OPTWAVE_RD"	Q 61.0	BOOL	// Signalband neues Design Farbe RD
"OX_GEN_OPTWAVE_GN"	Q 61.2	BOOL	// Signalband neues Design Farbe GN
"OX_GEN_OPTWAVE_BU"	Q 61.3	BOOL	// Signalband neues Design Farbe  BU
"OX_CU_FLUSH_JETS_ON"	Q 61.6	BOOL	// Ansteuerung Spuelung Spruehsystem
"OX_CU_FLUSH_ROOF_ON"	Q 61.7	BOOL	// Ansteuerung Spuelung Dach
"OX_TP_CALIBRATION_EXTEND"	Q 64.0	BOOL	// Messeinrichtung Messtaster ausfahren
"OX_TP_CALIBRATION_RUN_IN"	Q 64.1	BOOL	// Messeinrichtung Messtaster einfahren
"OX_TP_CALIBRATION_CLEAN"	Q 64.2	BOOL	// Messeinrichtung Messtaster abblasen
"OX_HCD_SST_CLAMP"	Q 65.0	BOOL	// Spannhydraulik Ruestplatz spannen
"OX_SP_HYD_RPL_SPANNDR_OK"	Q 65.1	BOOL	// Spannvorrichtung Spanndruck vorhanden
"OX_HCD_SST_UNPRESS"	Q 65.2	BOOL	// Ruestplatz Ventil Drucklos
"OX_SP_RPL_KUPPELN"	Q 67.0	BOOL	// Medienkupplung Ruestplatz einfahren
"OX_HCD_MACHINE_UNLOAD"	Q 67.1	BOOL	// Rueckmeldung Maschine Entladen
"OX_HCD_MPL_PRESSURE_OK"	Q 67.2	BOOL	// Spannvorrichtung Maschine gespannt
"OX_SP_SCH_SPANNVOR"	Q 67.3	BOOL	// Schmierstoffpumpe Spannfutter Spannvorrichtung
"OX_PW_RPL_PAL_KLEMMEN"	Q 68.0	BOOL	// Ruestplatz Palettenklemmung klemmen
"OX_PW_RPL_PAL_LOESEN"	Q 68.1	BOOL	// Ruestplatz Palettenklemmung loesen
"OX_SPI_TL_CLP_CLAMP"	Q 73.0	BOOL	// Werkzeugspanner spannen
"OX_TC_TL_BRUSH_CLEAN"	Q 73.1	BOOL	// Antrieb Buerste Reinigung Werkzeugkegel
"OX_GEN_POWERSAVE_N"	Q 97.0	BOOL	// Maschinenabschaltung
"OX_GEN_M_FUNCTION_M80"	Q 105.0	BOOL	// M-Funktionen M80
"OX_GEN_M_FUNCTION_M81"	Q 105.1	BOOL	// M-Funktionen M81
"OX_GEN_M_FUNCTION_M82"	Q 105.2	BOOL	// M-Funktionen M82
"OX_GEN_M_FUNCTION_M83"	Q 105.3	BOOL	// M-Funktionen M84
"OX_GEN_M_FUNCTION_M84"	Q 106.0	BOOL	// M-Funktionen M84
"OX_GEN_M_FUNCTION_M85"	Q 106.1	BOOL	// M-Funktionen M85
"OX_GEN_M_FUNCTION_M86"	Q 106.2	BOOL	// M-Funktionen M86
"OX_GEN_M_FUNCTION_M87"	Q 106.3	BOOL	// M-Funktionen M87
"OX_GEN_M_FUNCTION_M88"	Q 107.0	BOOL	// M-Funktionen M88
"OX_GEN_M_FUNCTION_M89"	Q 107.1	BOOL	// M-Funktionen M89
"OFX_GEN_EMSTP_CH1_N"	Q 110.0	BOOL	// Not-Aus Drehzahl
"OFX_GEN_STOP_CH1_MONITOR"	Q 110.1	BOOL	// Stillstandueberwachung
"OX_AL_Tempkomp_DSR"	Q 110.2	BOOL	// TEMPERATURKOMPENSATION: rücksetzen Synchronisation Temperaturdaten
"OX_AL_Tempkomp_CTS"	Q 110.3	BOOL	// TEMPERATURKOMPENSATION: Temperaturdaten auslesen
"OX_GEN_M_FUNCTION_M20"	Q 111.0	BOOL	// M-Funktionen M190
"OX_WM_WZ_STAT_einlegen"	Q 111.2	BOOL	// WZV: Lampe TIN (Werkzeug einlegen)
"OX_WM_WZ_STAT_entnehmen"	Q 111.3	BOOL	// WZV: Lampe TOUT  (Werkzeug entnehmen)
"OX_SH_HORIZONTAL_SWIVEL"	Q 112.0	BOOL	// Schwenkfraeskopf waagrecht M53
"OX_SH_VERTICAL_SWIVEL"	Q 112.1	BOOL	// Schwenkfraeskopf senkrecht M54
"OX_PS_DREHST_BREMSE_AUF"	Q 140.0	BOOL	// Achse 9 (Palettenrundspeicher)  Bremse lüften
"OX_PS_ABZIEHS_BREMSE_AUF"	Q 140.1	BOOL	// Bremse Kette 1 Palettenspeichersystem
"OX_PS_RPL_BREMSE_AUF"	Q 141.0	BOOL	// Bremse Rüstplatz lüften
"OX_PS_TURN_STATION_DOWN"	Q 142.0	BOOL	// Ventil Dreheinheit nach unten
"OX_PS_TURN_STATION_UP"	Q 142.1	BOOL	// Ventil Dreheinheit nach oben
"OX_PS_SST_DOOR_FRT_UNLOC"	Q 143.0	BOOL	// Ruestplatztuer vorn entriegeln
"OX_PS_SST_DOOR_RER_UNLOC"	Q 143.1	BOOL	// Ruestplatztuer hinten entriegeln
"OX_MI_TURNT_LUB_PUMP_ON"	Q 151.1	BOOL	// Schmierstoffpumpe ein Fraes-Drehtisch
"OX_U_AXIS_POSITION_0"	Q 170.0	BOOL	// U-Achse Position 0
"OX_U_AXIS_AXIS_OPER"	Q 170.1	BOOL	// U-Achse Betrieb
"OX_U_AXIS_CONFIRM_ALARM"	Q 170.2	BOOL	// U-Achse Quittierung Alarm
"OX_U_AXIS_PARK"	Q 170.3	BOOL	// U-Achse Park
"OX_U_AXIS_HEAD_EXIST"	Q 171.0	BOOL	// U-Achse Werkzeug angebaut
"OX_U_AXIS_CONTROL_ENABLE"	Q 171.1	BOOL	// U-Achse Reglerfreigabe
"OX_U_AXIS_EM_AX_OP"	Q 171.2	BOOL	// U-Achse Not-Achsbetrieb
"OX_TM_TOOL_CYL_LOCK"	Q 1000.1	BOOL	// Pneumatikzyl. Verriegelung WZ klemmen
"OX_TM_TOOL_CYL_UNLOCK"	Q 1000.2	BOOL	// Pneumatikzylinder Verriegelung Werkzeug loesen
"OX_PW_Freigabe"	Q 1000.3	BOOL	// Anforderung Freigabe Palettenwechsel
"OX_TC_CYL_1_TOOL_MAG"	Q 1001.1	BOOL	// Werkzeugmagazin Zylinder1 Richtung Magazin
"OX_TM_COUNTCLOCKWISE"	Q 1002.1	BOOL	// Werkzeugmagazin Linkslauf
"OX_TM_CLOCKWISE"	Q 1002.2	BOOL	// Werkzeugmagazin Rechtslauf
"OX_CA_MALFUNCT"	Q 1002.3	BOOL	// Kuehlaggregat Störmeldung Prioritaet 1
"OX_PC_CL_PRESS_HYD_OFF"	Q 1002.4	BOOL	// MA H4-03.7 Spannvorrichtung Verriegelung Palettenwechs
"OX_CA2_MALFUNCT"	Q 1002.5	BOOL	// Kuehlaggregat 2 Störmeldung Prioritaet 1
"OX_DH_CLAMP_RELEASE"	Q 1002.6	BOOL	// Klemmung loesen NC-Teilapparat
"OX_SP_HYD_EIN"	Q 1002.7	BOOL	// Spannhydraulik Pumpe ein
"OX_SP_HYD_RPL_LOESEDR_OK"	Q 1003.0	BOOL	// Spannvorrichtung Loesedruck vorhanden
"OX_KM_Motor_Kratzfoerd"	Q 1004.0	BOOL	// Antrieb Kratzerfoerderer
"OX_TM_TPU_GET_TOOL"	Q 1005.0	BOOL	// Transporteinheit auf Werkzeugkegel fahren
"OX_TM_TPU_RELEASE_TOOL"	Q 1005.1	BOOL	// Transporteinheit vom Werkzeugkegel wegfahren
"OX_TM_TPU_TRANSFERPOS"	Q 1005.2	BOOL	// Transporteinheit zu Übergabeposition fahren
"OX_TM_TPU_MAGAZINPOS"	Q 1005.3	BOOL	// Transporteinheit zur Magazinposition fahren
"OX_TM_MAG_TOOL_UNLOCK"	Q 1005.4	BOOL	// Werkzeug an Magazinposition entriegeln
"OX_TM_MAG_TOOL_LOCK"	Q 1005.5	BOOL	// Werkzeug an Magazinposition verriegeln
"OX_TM_TPU_AIR_CLEANING"	Q 1005.6	BOOL	// Druckluftreinigung der Transporteinheit einschalten
"OX_TM_TLOAD_TOOL_UNLOCK"	Q 1005.7	BOOL	// Werkzeug am Rüstplatz entriegeln
"OX_TM_TLOAD_TOOL_LOCK"	Q 1006.0	BOOL	// Werkzeug am Rüstplatz verriegeln
"OX_TM_RELEASE"	Q 1006.1	BOOL	// Werkzeugmagazin freigeben
"OX_TM_TLOAD_TOUT_H"	Q 1006.2	BOOL	// Meldung Werkzeug entnehmen
"OX_TM_TLOAD_TIN_H"	Q 1006.3	BOOL	// Meldung Werkzeug einlegen
"OX_TM_TLOAD_WDOW_UNLOCK"	Q 1006.4	BOOL	// Fenster Rüstplatz entriegeln
"OX_TC_MAGAZINPOS"	Q 1006.5	BOOL
"OX_TC_SPIPOS"	Q 1006.6	BOOL
"OX_KM_SPRUEHPIST_RPL_EIN"	Q 1009.0	BOOL	// Signalleuchte Spülpistole Rüstplatz Ein
"OX_PW_RPL_BREMSE_AUF"	Q 1009.1	BOOL	// Bremse NC-Ruestplatz Auf
"OX_SST_ENABLE_ROTATE"	Q 1009.2	BOOL	// Freigabe NC-Ruestplatz
"OX_SP_MPL_ENTKUPPELN"	Q 1016.0	BOOL	// SpannHydraulik Maschinenplatz entkuppeln
"OX_SP_MPL_KUPPELN"	Q 1016.1	BOOL	// SpannHydraulik Maschinenplatz kuppeln
"OX_SO_WFK_UMSCH_KM"	Q 1016.5	BOOL	// Wiegenfräskopf Kühlmittel Umschaltung
"OX_KM_SF_KRATZER_EIN_V"	Q 1017.0	BOOL	// Antrieb Kratzerförderer „Ein“
"OX_KM_SF_HEBEPUMPE_EIN"	Q 1017.1	BOOL	// Hebepumpe Schmutztank „Ein“
"OX_AL_Messsignal_Umsch"	Q 1017.2	BOOL	// Umschaltung Messsignale MesstasterTS27 / Laser
"OX_TT_ausschwenken"	Q 1017.3	BOOL	// Messtaster Tisch TS27R ausschwenken
"OX_TT_einschwenken"	Q 1017.4	BOOL	// Messtaster Tisch TS27R einschwenken
"OX_PW_HUB_2_HEBEN"	Q 1019.0	BOOL	// Palettenwechsler Hubeinheit nach oben schnell
"OX_PW_HUB_2_SENKEN"	Q 1019.1	BOOL	// Palettenwechsler Hubeinheit nach unten schnell
"OX_PC_MPL_PALLET_MONITOR"	Q 1020.0	BOOL	// Druckluft Palettenerkennung
"OX_TLB_CLEAN"	Q 1020.1	BOOL	// Blasluft Werkzeugbruchueberwachung
"OX_PC_VALVE_REQUEST"	Q 1020.2	BOOL	// Palettenwechsler Ventilabfrage Luftstrom Palette
"OX_FMS_OM1_DISABLED"	Q 1027.0	BOOL	// Betriebsart Automatik gesperrt Palettenspeichersystem
"OX_ROBOT_COP1"	Q 1028.0	BOOL	// Freigabe Spannfutter
"OX_ROBOT_DOOR_CLOSE"	Q 1028.1	BOOL	// Hubtuere Werkstuecklader schliessen
"OX_ROBOT_DOOR_OPEN"	Q 1028.2	BOOL	// Hubtuere Werkstuecklader oeffnen
"OX_ROBOT_START"	Q 1028.3	BOOL	// Startsignal Werkstueckwechsel Handlingsystem
"OX_ROBOT_TCP1"	Q 1028.4	BOOL	// Freigabe Werkstueckwechsel
"OX_WA_REQUEST_DOOR_UNLOC"	Q 1028.5	BOOL	// Anforderung Kabinentuer entriegeln
"OX_HCD_TST_MCON_CLEAN"	Q 1034.0	BOOL	// Hydraulik Maschinenplatz Kupplung abblasen   /H4-08.2
"OX_HCD_SST_BLOW_AIR"	Q 1034.2	BOOL	// Medienkupplung Ruestplatz abblasen
"OX_HCD_ON"	Q 1034.3	BOOL	// Spannhydraulik ein   /H4-01.6
"OX_TP_ENABLE"	Q 1051.0	BOOL	// Startsignal Messtaster
"OX_SO_WFK_KLE_KLEMMEN"	Q 1051.1	BOOL	// Wiegenfräskopf Klemmung klemmen
"OX_SO_WFK_KLE_LOESEN"	Q 1051.2	BOOL	// Wiegenfräskopf Klemmung lösen
"OX_SO_WFK_MEDIENK_REINIG"	Q 1051.3	BOOL	// Wiegenfräskopf Medienkupplung abblasen/reinigen
"OX_SO_WFK_PNEUMATIK_EIN"	Q 1051.4	BOOL	// Wiegenfräskopf Pneumatik Ein
"OX_SO_DMS_PNEUMAK_EIN"	Q 1051.5	BOOL	// Drehmomentstütze Pneumatikversorgung Ein
"OX_PC_MPL_MCON_DISENGAGE"	Q 1051.6	BOOL	// Medienkupplung Fraes-Drehtisch einfahren
"OX_PC_MPL_MCON_ENGAGE"	Q 1051.7	BOOL	// Medienkupplung Fraes-Drehtisch ausfahren
"OX_PW_SCH_PUMPE_EIN"	Q 1052.0	BOOL	// Schmierung Palettenwechsler
"OX_SP_H_SPANNSTELLE_1"	Q 1053.0	BOOL	// Spannhydraulik Lampe Spannstelle 1
"OX_SP_H_SPANNSTELLE_2"	Q 1053.1	BOOL	// Spannhydraulik Lampe Spannstelle 2
"OX_SP_H_SPANNSTELLE_3"	Q 1053.2	BOOL	// Spannhydraulik Lampe Spannstelle 3
"OX_SP_H_SPANNSTELLE_4"	Q 1053.3	BOOL	// Spannhydraulik Lampe Spannstelle 4
"OX_SP_RPL_AUFL_ENTSPAN"	Q 1053.4	BOOL	// Ventil Luft für Auflagenkontrolle gelöst am Rüstplatz
"OX_SP_RPL_AUFL_SPANNEN"	Q 1053.5	BOOL	// Ventil Luft für Auflagenkontrolle gespannt am Rüstplatz
"OX_SP_RPL_BLASLUFT"	Q 1053.6	BOOL	// Ventil Luft für Vorrichtung Abblasen
"OX_SP_RPL_MPL_BLASLUFT"	Q 1053.7	BOOL	// Ventil Blasluft Medienkupplung
"OX_RELEASEUNI_GET_TOOL"	Q 1054.0	BOOL	// Ausrückstation Hub Richtung Werkzeugkegel
"OX_RELEASEUNI_RELEASE_T"	Q 1054.1	BOOL	// Ausrückstation Hub in Grundstellung
"OX_RELEASEUNI_TRANSPOS"	Q 1054.2	BOOL	// Ausrückstation Hub Richtung Übergabeposition
"OX_RELEASEUNI_MAGAZINPOS"	Q 1054.3	BOOL	// Ausrückstation Richtung Magazinposition
"OX_RELU_MAG_TOOL_UNLOC"	Q 1054.4	BOOL	// Ausrückstation WZ Greifer entriegeln
"OX_RELU_TST_TOOL_UNLOC"	Q 1054.5	BOOL	// Ausrückstation WZ-Pin Magazinplatz entriegeln
"OX_RELU_TOOL_C_BL_AI"	Q 1054.6	BOOL	// Ausrückstation Blasluft Kegel- und Sensorreinigung
"OX_CU_FLUSCH_PUMP_PC"	Q 1054.7	BOOL	// Klauenspülung während PW ein
"OX_HCD_MPL_ENGAGE"	Q 1061.0	BOOL	// Hydraulik Maschinenplatz Kupplung ankuppeln   /H4-05.3
"OX_HCD_MPL_DISENGAGE"	Q 1061.1	BOOL	// Hydraulik Maschinenplatz Kupplung abkuppeln   /H4-05.3
"OX_HCD_SST_ENGAGE"	Q 1061.2	BOOL	// Hydraulik Rüstplatz Kupplung ankuppeln   /H4-06.3
"OX_HCD_SST_DISENGAGE"	Q 1061.3	BOOL	// Hydraulik Rüstplatz Kupplung abkuppeln   /H4-06.3
"OX_HCD_LUB_ON"	Q 1061.4	BOOL
"OX_HCD_SST_PRESSURE_OFF"	Q 1061.5	BOOL
"OX_VMS_MSG_BEA_START"	Q 1062.0	BOOL
"OX_VMS_MSG_FPRINT_START"	Q 1062.1	BOOL	// IFM-Vibrationsüberwachung Fingerprint-Messung starten
"OX_PC_ENABLE"	Q 1062.5	BOOL	// Anforderung Freigabe Palettenwechsler   /G1-05.4
"OX_HCD_CL_PR_SST_CLPED_H"	Q 1062.6	BOOL	// Spannhydraulik Leuchtmelder Vorrichtung spannen   /H4-10.3
"OX_HCD_CL_PR_SST_RELD_H"	Q 1062.7	BOOL	// Spannhydraulik Leuchtmelder Vorrichtung entspannen   /H4-10.6
"OX_SP_RPL_ENTKUPPELN"	Q 1067.1	BOOL	// Medienkupplung Ruestplatz ausfahren
"OX_WK_ZYL_1_AUSF"	Q 1067.2	BOOL	// Werkzeugträger Zylinder 1 ausfahren
"OX_WK_ZYL_1_EINFAHREN"	Q 1067.3	BOOL	// Werkzeugträger Zylinder 1 einfahren
"OX_WK_ZYL_2_AUSF"	Q 1067.4	BOOL	// Werkzeugträger Zylinder 2 ausfahren
"OX_WK_ZYL_2_EINFAHREN"	Q 1067.5	BOOL	// Werkzeugträger Zylinder 2 einfahren
"OX_WK_KLAPPE_AUF"	Q 1067.6	BOOL	// Werkzeugklappe oeffnen
"OX_WK_KLAPPE_ZU"	Q 1067.7	BOOL	// Werkzeugklappe schliessen
"OX_PC_SST_PALLET_RELEASE"	Q 1077.0	BOOL	// Ruestplatz Palettenklemmung loesen   /G1-35.4
"OX_PC_SST_PALLET_CLAMP"	Q 1077.1	BOOL	// Ruestplatz Palettenklemmung klemmen   /G1-35.4
"OX_HCD_SST_CL_PO_1_SEL_H"	Q 1078.4	BOOL	// Spannhydraulik Rüstplatz Leuchtmelder Spannstelle 1 aktiv   /H4-50.3
"OX_HCD_SST_CL_PO_2_SEL_H"	Q 1078.5	BOOL	// Spannhydraulik Rüstplatz Leuchtmelder Spannstelle 2 aktiv   /H4-50.6
"OX_CC_RAKE_1_FORWARD"	Q 1081.0	BOOL	// Spaenefoerderer- Rechen 1 Hubeinheit vor
"OX_CC_RAKE_1_BACKWARD"	Q 1081.1	BOOL	// Spaenefoerderer- Rechen 1 Hubeinheit zurueck
"OX_CC_RAKE_2_FORWARD"	Q 1081.2	BOOL	// paenefoerderer- Rechen 2 Hubeinheit vor
"OX_CC_RAKE_2_BACKWARD"	Q 1081.3	BOOL	// Spaenefoerderer- Rechen 2 Hubeinheit zurueck
"OX_CC_RAKE_M_VALVE"	Q 1081.4	BOOL	// Ventil Hauptluft Spaenefoerderer-Rechen
"OX_FMS_PALLET_ON_APC"	Q 1150.1	BOOL	// MC OUTPUT Byte 1 Bit 1
"OX_FMS_CRANE_MOVE_OK"	Q 1150.2	BOOL	// MC OUTPUT Byte 1 Bit 2
"OX_FMS_APC_A_SIDE_OUT"	Q 1150.3	BOOL	// MC OUTPUT Byte 1 Bit 3
"OX_FMS_APC_B_SIDE_OUT"	Q 1150.4	BOOL	// MC OUTPUT Byte 1 Bit 4
"OX_FMS_PALLET_CHANGE_AKT"	Q 1150.5	BOOL	// MC OUTPUT Byte 1 Bit 5
"OX_FMS_APC_DOOR_CLOSED"	Q 1150.6	BOOL	// MC OUTPUT Byte 1 Bit 6
"OX_FMS_OM_ENABLE"	Q 1150.7	BOOL	// MC OUTPUT Byte 1 Bit 7
"OX_FMS_MACHINE_PGM_RUN"	Q 1151.0	BOOL	// MC OUTPUT Byte 2 Bit 0
"OX_FMS_CUTTING"	Q 1151.1	BOOL	// MC OUTPUT Byte 2 Bit 1
"OX_FMS_MACHINE_ERROR"	Q 1151.2	BOOL	// MC OUTPUT Byte 2 Bit 2
"OX_FMS_FIXTURE_EXIST"	Q 1151.3	BOOL	// MC OUTPUT Byte 2 Bit 3
"OX_FMS_FIXTURE_RELEASED"	Q 1151.4	BOOL	// MC OUTPUT Byte 2 Bit 4
"OX_GEN_OM_ID_DATA_0"	Q 1151.5	BOOL	// Smartkey: Rückmeldung Daten – Spur 1
"OX_GEN_OM_ID_DATA_1"	Q 1151.6	BOOL	// Smartkey: Rückmeldung Daten – Spur 2
"OX_SPI_IMP_DELETE"	Q 2030.0	BOOL	// Impuls Hauptantrieb geloescht (55/65H)
"OX_INFEED_ENABLE_NCU"	Q 2030.1	BOOL	// Ansteuerung NCU: Freigabe Klemme X122.1 SLM bereit (55/65H)
"OX_ENABLE_OUT_3_NX_NCU"	Q 2030.2	BOOL	// Ansteuerung NCU: Freigabe Klemme X122.2 AUS3 (55/65H)
"OX_INFEED_ENABLE_NX"	Q 2030.3	BOOL	// Ansteuerung NX: Freigabe Klemme X122.1 Einspeisung ok (55/65H)
"OX_CU_GAP_SCREEN_CLEAN"	Q 2030.4	BOOL	// Kühlmittelanlage Spaltsieb ein / nach oben  (55/65H)
"OX_TM_PUMP"	Q 2030.5	BOOL	// Hebepumpe Werkzeugmagazin (55/65H)
"OX_CU_FLUSH_PIST_SST_ON"	Q 2030.6	BOOL	// Meldung Spuelpistole Ruestplatz ein
"OX_TC_ENABLE_BRUSH_CLEAN"	Q 2030.7	BOOL	// Freigabe Positionierung Reinigung
"OX_TORQ_PROP_CAIR_ON"	Q 2031.0	BOOL	// Blasluft Drehmomentstuetze
"BT_ET200S_4_14"	Q 3030.0	BOOL	// Reserve Modul
"OX_SST_FLUSH_ON_H"	Q 3046.2	BOOL	// B2-87.6 Ruestplatz Spuelung aktiv (Meldeleuchte)
"OX_SST_SC_CL_PO_1_STATE"	Q 3070.0	BOOL	// H4-93.2 Status Auflagenkontrolle Spannstelle 1 (Meldeleuchte)
"OX_SST_SC_CL_PO_2_STATE"	Q 3070.1	BOOL	// H4-93.4 Status Auflagenkontrolle Spannstelle 2 (Meldeleuchte)
"OX_SST_FIXT_CL_PO_1_CLE"	Q 3093.2	BOOL	// H4-94.2 Auflagenkontrolle Luft für Reinigung (hoher ALK-Druck)
"OX_SST_SC_SENS_ACT"	Q 3093.3	BOOL	// H4-94.4 Auflagenkontrolle Luft für Messung (niedriger ALK-Druck)
"OW_VMS_SPI_SPEED_RPM"	QW 1048	WORD
"OW_CU_SET_VAL_PRESSURE"	QW 1600	WORD	// Kühlmittel Hochdruck PROP-Ventil
"SET_CLK"	SFC 0	SFC 0	// Set System Clock
"READ_CLK"	SFC 1	SFC 1	// Read System Clock
"GADR_LGC"	SFC 5	SFC 5	// Query Logical Address of a Channel
"RD_SINFO"	SFC 6	SFC 6	// Read OB Start Information
"D_ACT_DP"	SFC 12	SFC 12	// Deactivating and Activating DP Slaves
"DPNRM_DG"	SFC 13	SFC 13	// Read Diagnostic Data of a DP Slave
"DPWR_DAT"	SFC 15	SFC 15	// Write Consistent Data to a Standard DP Slave
"ALARM_SQ"	SFC 17	SFC 17	// Generate Block-Related Messages with Acknowledgment
"BLKMOVE"	SFC 20	SFC 20	// Block move
"FILL"	SFC 21	SFC 21	// Initialize a Memory Area
"CREAT_DB"	SFC 22	SFC 22	// Create Data Block
"UPDAT_PI"	SFC 26	SFC 26	// Update Process Image Input
"SET_TINT"	SFC 28	SFC 28	// Set Time-of-Day Interrupt
"CAN_TINT"	SFC 29	SFC 29	// Cancel Time-of-Day Interrupt
"ACT_TINT"	SFC 30	SFC 30	// Activate Time-of-Day Interrupt
"DIS_AIRT"	SFC 41	SFC 41	// Delay the Higher Priority Interrupts and Asynchronous Errors
"EN_AIRT"	SFC 42	SFC 42	// Enable Higher Priority Interrupts and Asynchronous Errors
"STP"	SFC 46	SFC 46	// Change the CPU to STOP
"WAIT"	SFC 47	SFC 47	// Delay Execution of the User Program
"LGC_GADR"	SFC 49	SFC 49	// Query the Module Slot Belonging to a Logical Address
"RD_LGADR"	SFC 50	SFC 50	// Read All Logical Addresses of a Module
"RDSYSST"	SFC 51	SFC 51	// Read a System Status List or Partial List
"WR_USMSG"	SFC 52	SFC 52	// Write a User-Defined Diagnostic Event to the Diagnostic Buffer
"TIME_TCK"	SFC 64	SFC 64	// Read the System Time
"T0_Siemens"	T 0	TIMER	// Timer für Siemens-Grundprogramm
"T1_Siemens"	T 1	TIMER	// Timer für Siemens-Grundprogramm
"T2_Siemens"	T 2	TIMER	// Timer für Siemens-Grundprogramm
"T3_Siemens"	T 3	TIMER	// Timer für Siemens-Grundprogramm
"T4_Siemens"	T 4	TIMER	// Timer für Siemens-Grundprogramm
"T5_Siemens"	T 5	TIMER	// Timer für Siemens-Grundprogramm
"T6_Siemens"	T 6	TIMER	// Timer für Siemens-Grundprogramm
"T7_Siemens"	T 7	TIMER	// Timer für Siemens-Grundprogramm
"T8_Siemens"	T 8	TIMER	// Timer für Siemens-Grundprogramm
"T9_Siemens"	T 9	TIMER	// Timer für Siemens-Grundprogramm
"Te_TempTransmitter_t10"	T 10	TIMER	// TEMPERATURKOMPENSATION:
"T11"	T 11	TIMER	// Reserve
"T12"	T 12	TIMER	// Reserve
"Ta_WM_Energiefreigabe"	T 13	TIMER	// Timer für WM-Energiefreigabe
"T14"	T 14	TIMER	// Reserve
"T15"	T 15	TIMER	// Reserve
"Tv_MinSchm_M7"	T 16	TIMER	// Minimalmengen Schmierung: Leitung bei M7 ausblasen
"T_MA_Timer_Hydraulik"	T 17	TIMER	// Timer HydraulikEin
"T_MA_Timer_Schmierung"	T 18	TIMER	// Timer Schmierung
"t_hyd_fuell_min_verz"	T 19	TIMER	// Hydraulik Füllstand Minimum verzögert
"T_Messdose_Bereit"	T 20	TIMER	// Messdose: Überwachung Bereitschaft
"Te_Spindel_Stop_"	T 21	TIMER	// Verzögerung Spindel Stop bei Alarm
"Te_Spindel_Stop_Geo"	T 22	TIMER	// Verzögerung Spindel Stop bei Alarm
"Te_SK_Ablauf"	T 23	TIMER	// SCHWENKKOPF:Timer Schwenkkopf Ablauf
"Te_SK_Entprellzeit"	T 24	TIMER	// SCHWENKKOPF:Timer Schwenkopf Entprellen
"Te_SK_FehlerUebw"	T 25	TIMER	// SCHWENKKOPF:Timer ScnkwenkkopfFehlerueberwachung
"TE_PW_Spuelung"	T 26	TIMER	// PW: Timer Spuelung
"Te_Mag_Zaehlimp"	T 27	TIMER	// GT MAG: Timer Zaehlimpulsüberwachung
"Te_Kmtl_Ueberlauf"	T 28	TIMER	// KMTL: Timer Ueberlauf
"T_Messwert_Intervall"	T 29	TIMER	// TEMPERATURKOMPENSATION: fc242
"TE_Blum_FehlUebw"	T 30	TIMER	// Laser: Zeitueberwachung Hub ausfahren
"Te_Ueb_WZW_HUB"	T 31	TIMER	// FC_UT_DYN_UEBW: Zeitzähler WZW HUB
"TE_Kalibr_FehlUebw"	T 32	TIMER	// Kalibrierring: Zeitueberwachung Hub ausfahren
"Tv_2Stufiges_Getr"	T 33	TIMER	// Getriebe: Timer Überwachung
"Te_AX_Mot_Temp"	T 34	TIMER	// AX: Not-Aus nach Motorübertemperatur
"Te_DrehDurch_Fuell"	T 35	TIMER	// DrehDurchführung Füllstandsüberwachung
"Te_AX_X_Bremse_loesen"	T 36	TIMER	// Timer Einschaltverzögert X-Achse: Bremse lösen
"Te_AX_Y_Bremse_loesen"	T 37	TIMER	// Timer Einschaltverzögert Y-Achse: Bremse lösen
"Te_AX_Z_Bremse_loesen"	T 38	TIMER	// Timer Einschaltverzögert Z-Achse: Bremse lösen
"Te_AX_A_Bremse_loesen"	T 39	TIMER	// Timer Einschaltverzögert 4-Achse: Bremse lösen
"Te_AX_B_Bremse_loesen"	T 40	TIMER	// Timer Einschaltverzögert 5/11-Achse: Bremse lösen
"Te_WZW_Ablauf"	T 41	TIMER	// WZW: Timer Ablauf
"T42"	T 42	TIMER	// Reserve
"Te_PW_GST_pruefen"	T 43	TIMER	// Palettenwechsler Grundstellung überprüfen
"Te_Tuer_zu"	T 44	TIMER	// MA: Timer Ueberwachung schliessen Tuerverriegelung
"Te_Verz_Leistung"	T 45	TIMER	// MA: Timer Verzoegerung Leistung ein
"Te_Uebw_ER-Modul"	T 46	TIMER	// MA: Timer für Überwachung ER-Modul
"TA_Spindel_Freischn"	T 47	TIMER	// SPINDEL: Timer zum Freischneiden
"T48"	T 48	TIMER	// Reserve
"TV_Spannvorrichtung"	T 49	TIMER	// Timer der Spannvorrichtung
"Te_FehlerQuit_Taste"	T 50	TIMER	// Verlängerung Quittiertaste
"Te_AX_7_Bremse_loesen"	T 51	TIMER	// Timer Einschaltverzögert AX 7-Achse: Bremse lösen
"Te_MagTuer_Ver"	T 52	TIMER	// Zeitverzögerung Verriegeln Tuer
"TE_RPL_ZH"	T 53	TIMER	// Rüstplatz-Achse Überwachungszeit Zweihandbedienung
"T_druckstufe"	T 54	TIMER	// Timer IKZ Druckstufe
"TV_BHG_Anz_Akt"	T 55	TIMER	// BHG Anzeige aktivieren verlängerter Impuls
"Ta_8.Achse_Bremse_auf"	T 56	TIMER	// Timer für 8.Achse Bremse öffnen
"TV_RPL_AX_IN_POS"	T 57	TIMER	// Rüstplatz-Achse Sollposition erreicht verlängerter Impuls
"TA_RPL_AX_FRG_BREMSRAMPE"	T 58	TIMER	// Rüstplatz-Achse Freigabe links / Rechts drehen (Bremsrampenzeit)
"TV_WZB_Abblastimer"	T 59	TIMER	// Werkzeugbruchüberwachung Abblaszeit
"Ta_RFGSpindelAbf_T60"	T 60	TIMER	// Reglerfreigabe Spindel abfallverzögert
"Te_Timer_RegFES"	T 61	TIMER	// Reglerfreigabe Spindel einschaltverzögert
"Te_Timer_Yd"	T 62	TIMER	// Stern Dreieck Timer
"Te_Timer_Uebw_Yd"	T 63	TIMER	// Stern Dreieck Überwachungstimer
"Te_WZW_Hub_Verz"	T 64	TIMER
"Ta_9.Achse_Bremse_auf"	T 65	TIMER	// Timer für 9.Achse Bremse öffnen
"Ta_Be_Entladen_aktiv"	T 66	TIMER
"Ta_Systemdruck"	T 67	TIMER	// Ausgang Druckluft Ein abfallverzögert
"T68"	T 68	TIMER	// Reserve
"Te_Entprell_sync"	T 69	TIMER	// Werkzeugmagazin: Enprellen Überwachung Synchronisation
"Te_Oelstand_Warnung"	T 70	TIMER	// SS: Timer Oelstand Spindelschmierung Warnung
"Te_Oelstand_Fehler"	T 71	TIMER	// SS: Timer Oelstand Spindelschmierung Fehler
"Te_Luftdruck_Warnung"	T 72	TIMER	// SS: Timer Luftdruck nicht 1 Warnung
"Te_Luftdruck_Fehler"	T 73	TIMER	// SS: Timer Luftdruck nicht 1 Fehler
"Te_Luftdrucknicht0"	T 74	TIMER	// SS:Timer für Luftdruck nicht 0 Warnung
"Tv_PS_RPL_entriegeln"	T 75	TIMER	// Palettenspeicher Rüstplatztüren Hinten+Vorne entriegeln
"Tv_Wzsp_Verzoegerung"	T 76	TIMER	// WSP: Timer fuer Werkzeugspanner Verzoegerung
"Tv_Ausgang_Spuelpistole"	T 77	TIMER	// SPP: Spuelpistolenausgang verzoegert abschalten
"Te_Spi_Temp_1"	T 78	TIMER	// SPINDEL:  Temperaturüberwachung_1
"Te_Spi_Eingang"	T 79	TIMER	// SPINDEL:  Spindeleingang entprellt überwacht
"t_verz_PW_unten_daten"	T 80	TIMER	// Verzoegerung Palettenwechsler unten wegen Daten umkopieren an Fastems
"TV_HR_Entprell"	T 81	TIMER	// Entprellen der Zustimmtaste BHG
"TE_RCKMLD_Druck0_OK"	T 82	TIMER	// Überwachungszeit Kühlmittelanlage Rückmeldung Druckstufe
"Te_PW_Palette_vorhanden"	T 83	TIMER	// Timer für Palette im Arbeitsraum vorhanden
"Te_PW_AX_Wechselpos"	T 84	TIMER	// Timer für Palettenwechsler-Achsen in Wechselposition
"t_verz_wzw_aktiv"	T 85	TIMER	// Verzögerung für Überwachung Werkzeugwechsel zu langsam/steht
"Te_Tsz"	T 86	TIMER	// Freigabe Palettenwechsel 0-Signal verzögert
"Te_Spi_Temp_2"	T 87	TIMER	// SPINDEL:  Temperaturüberwachung_2
"Te_Ende_SpNachschm"	T 88	TIMER	// Freigabe Kühlmittelanlage von PNOZ fehlt verzögert
"Te_PIN_LOCKED"	T 89	TIMER	// Verzögerung der Abfrage ob PINLOCK verriegelt
"Tv_Ax4_Klemmung"	T 90	TIMER	// AX: Verzoegerungszeit im Rundachsmodul Achse 4
"Tv_Ax5_Klemmung"	T 91	TIMER	// AX: Verzoegerungszeit im Rundachsmodul Achse 5/11
"Tv_Ax4_Fehl_Ueb"	T 92	TIMER	// AX: Fehlerüberwachung Achse 4
"Tv_Ax5_Fehl_Ueb"	T 93	TIMER	// AX; Fehlerüberwachung Achse 5/11
"Te_Mag_ZH"	T 94	TIMER	// Überwachungszeit Zweihandbedienung Werkzeugmagazin
"Te_Energ_ZH"	T 95	TIMER	// Externe Energiefreigabe Werkzeugmagazin verzögert
"Te_Verz_DL_Ueberw"	T 96	TIMER	// Pneumatikdruck ist 0 Signal verzögert
"Tv_Messtater_aktiv"	T 97	TIMER	// Messtaster aktiv verzögert
"T_WZB"	T 98	TIMER	// Timer Werkzeugbruchüberwachung
"T_VERZ_ABFR_MPL_BELEGT"	T 99	TIMER	// Werkzeugregal Abfrage Magazinplatz belegt verzögert
"Tv_Reset_Impuls"	T 100	TIMER	// MA: Reset Impuls verlängert
"Tv_Messtaster_Trigger"	T 101	TIMER	// MESS:Nachtrigern des Messtasters nach 45 sec
"Tv_Messtaster_Blasluft"	T 102	TIMER	// MESS:Messtaster Blasluft ansteuern mit M26
"Tv_Messtaster_Fehler"	T 103	TIMER	// MESS:Messtaster Überwachung Bereitschaftsignal
"T104"	T 104	TIMER	// T104
"T105"	T 105	TIMER	// T105
"Te_I_PW_MPL_MDK_GEKUPP"	T 106	TIMER	// Medienkupplung Fraes-Drehtisch ausgefahren verzögert
"Te_Fehler_ASUP_M5"	T 107	TIMER	// ASUP: Fehlerüberwachung M5 TempKomp
"Te_I_PW_MPL_MDK_ENTKUPP"	T 108	TIMER	// Medienkupplung Fraes-Drehtisch eingefahren verzögert
"Ta_Schmierluftaus"	T 109	TIMER	// Schmierluftventil ein abfallverzögert
"TA_WZW_SUCHEN_U_POSITION"	T 110	TIMER	// WZW: MAG verfahren über Suchen & Positionieren  bzw. Taste -> T-Befehl sperren
"Ti_Init_Maschine"	T 111	TIMER	// ASUP: Verriegeln Reset bei Initialisierungs-Asups
"Tv_ResetTaste_WZV_verr"	T 112	TIMER	// ResetTaste verzögern bei anst. Auftrag
"Tv_ResetTaste_WZV_verl"	T 113	TIMER	// Reset Taste bei quittiertem Auftrag bringen
"Te_KegRein"	T 114	TIMER	// FC_UT_DYN_UEBW : Zeitzähler WZW Kegelreinigung
"Te_Verrieg"	T 115	TIMER	// FC_UT_DYN_UEBW : Zeitzähler WZW Verriegelung
"Te_Papierband_ende"	T 116	TIMER	// Kühlmittelanlage Papierband Ende
"T1_DynUebw_Zeitzaehler"	T 117	TIMER	// FC_UT_DYN_UEBW : Zeitzähler WZW Überwachung Bruch
"Te_PWKlemmbd1Signal"	T 118	TIMER	// Eingänge Klemmung Palettenwechsler beide 1-Signal verzögert
"Ta_sperre_T_Aufruf"	T 119	TIMER	// Nächsten T-Befehl sperren abfallverzögert
"Te_Achs14"	T 120	TIMER	// Timer Einschaltverzögert AX 14-Achse: Bremse lösen
"T_DREHZAHL_OK"	T 121	TIMER
"Timer_Req_SPI_DATA"	T 122	TIMER	// Vibrationssensor Anforderung Spindeldaten
"T_HAX_Stehen"	T 123	TIMER
"T_LS_FehlerUebw"	T 124	TIMER	// Palettenspeicher Überwachungszeit Bewegungen
"Te_LS_Entprellzeit"	T 125	TIMER	// Palettenspeicher Entprellzeit
"Te_AX12_BremseLoes"	T 126	TIMER	// Timer Einschaltverzögert AX...-Achse: Bremse lösen
"Te_FM_WW_Teller"	T 127	TIMER	// Verzögerte Fehlermeldungen Werkzeugwechsel Teller
"T_FD_SCHMIERSTAND"	T 128	TIMER	// Fräs-Drehtisch Schmierung: Füllstand nicht ok verzögert
"T_FD_RUECKM_SCHMIE"	T 129	TIMER	// Fräs-Drehtisch Schmierung: Überwachungzeit HUB Schmierimpuls
"T2_DynUebw_Zeitzaehler"	T 130	TIMER	// FC_UT_DYN_UEBW : Zeitzähler WZW Pneumatische Greiferentriegelung Greifer 2
"Te_Grf2_Verriegelung"	T 131	TIMER	// Greifer 2 verriegelt verzögert
"Ta_DP_Diagnose"	T 132	TIMER	// Profibus-Einzel-Diagnose
"T_verz_PW_JOB"	T 133	TIMER	// Palettenwechsler Jobbetrieb verzögert
"TE_Hpt_Achsen_Stehen"	T 134	TIMER	// Gesamt Vorschub Halt Hauptachsen verzögert
"TE_WZW_aktiv_gewesen"	T 135	TIMER	// Werkzeugwechsel aktiv abfallverzögert
"Te_Meldung_Jobliste"	T 136	TIMER	// Kein Job gefunden oder kein Rohteil vorhanden verzögert
"T_TPF_Motor_Ein"	T 137	TIMER	// Kühlmittelanlage Papierbandfilter ein verzögert
"Tv_Ax6_Klemmung"	T 138	TIMER	// AX: Verzoegerungszeit im Rundachsmodul Achse 6 (Spindel)
"Tv_Ax6_Fehl_Ueb"	T 139	TIMER	// AX: Fehlerüberwachung Achse 6 (Spindel)
"T_Temp_read_ok"	T 140	TIMER	// TEMPERATURKOMPENSATION: lesen fertig
"Te_Ueb_WZW_Tuer"	T 141	TIMER	// FC_UT_DYN_UEBW : Zeitzähler WZW Türe
"Te_Greifer"	T 142	TIMER	// FC_UT_DYN_UEBW : Zeitzähler WZW Greifer
"T_Tüere_entr_bei_ZD"	T 143	TIMER	// Timer bei ZD muß Tür-Taste langer betätigt werden
"Te_KM_MAX_NIVEAU"	T 144	TIMER	// Kühlmittelanlage: Maximaler Füllstand überschritten verzögert
"Te_RS_Uebw_RP"	T 145	TIMER	// Rüstplatztüre Zu/Verriegelt Überwachungszeit
"Ta_RS_Tuer_Verr"	T 146	TIMER	// Rüstplatztüre verriegeln abfallverzögert
"Te_Achs8"	T 147	TIMER	// Timer Einschaltverzögert AX 8-Achse: Bremse lösen
"Te_Achs9"	T 148	TIMER	// Timer Einschaltverzögert AX 9-Achse: Bremse lösen
"Te_Achs10"	T 149	TIMER	// Timer Einschaltverzögert AX 10-Achse: Bremse lösen
"TV_Vorwarnung_KMTL"	T 150	TIMER	// Kühlmittelanlage: Vorwarnung Kühlmittelmangel verzögert
"Tv_OENEB_NAchlZ"	T 151	TIMER	// Oel-Nebelabscheider Nachlaufzeit
"T_Kratzfoerderer"	T 152	TIMER	// KMTL: Kratzförderer Nachlaufzeit
"Tv_KM_TPFMOTOR_EIN"	T 153	TIMER	// Timer für  O_KM_TPF_MOTOR_EIN
"Te_RP_4s_entriegelt"	T 154	TIMER	// Rüstplatztüre entriegeln verzögern
"Te_Ueberw_Drehdurchführ"	T 155	TIMER	// Überwachungszeit Leckage Drehdurchführung
"T_Trigger_HaSyst"	T 156	TIMER
"Ta_WZ_ablegen_aktiv"	T 157	TIMER	// Werkzeug ablegen aktiv abfallverzögert
"T_SPL_AKTIV"	T 158	TIMER	// FRÄS-DREHTISCH SCHMIERUNG: Zyklenschalter Progressivverteiler verzögert
"Ta_T_Prepare_aktiv"	T 159	TIMER	// Werkzeug Vorbereitung aktiv abfallverzögert
"Te_Rein_Fuell_Max"	T 160	TIMER	// KMTL: Überlauf Kühlmittel Grobbereich verzögert
"Tv_nEintr"	T 161	TIMER	// SV an SOKO: neuer Alarmeintrag erfolgt
"Te_SpiKlemm_beide_1Signa"	T 162	TIMER	// Eingänge Klemmung Spindel beide 1-Signal verzögert
"Tv_FM_Hawe_unterdruecken"	T 163	TIMER	// FM-Hawe: Druck nicht erreichbar verzögert auswerten
"T_FD_SCHMIER_WAR"	T 164	TIMER
"Te_13te_Achs_Bremse_löse"	T 165	TIMER	// Timer Einschaltverzögert 13-Achse: Bremse lösen
"T_wgfTUe"	T 166	TIMER	// Wzw.Grundstellung fahren Schritt Überwachungszeit
"Te_Stoer_Nebelabscheider"	T 167	TIMER	// Oel-Nebelabscheider Störung verzögert
"Te_Diagnoseschalter"	T 168	TIMER	// Kühlmittelanlage: Diagnose verzögert
"TV_M190"	T 169	TIMER	// Zusatzfunktion M190 verzögert
"Tv_JOB_sperr"	T 170	TIMER	// Timer für Signal JOB_sperr
"Te_Prg_nicht_aktiv_ASUP"	T 171	TIMER	// TE: Programm nicht aktiv für ASUP-Start
"Te_Spanner_nicht_geloest"	T 172	TIMER	// Überwachungszeit Werkzeugspanner gelöst
"TE_SPA_schlies_Taste"	T 173	TIMER	// Überwachungszeit Werkzeugspanner gespannt
"Verz_Abfrage_inPos"	T 174	TIMER	// Befehl Magazin positionieren verzögert
"T_SA_HW_Test_laeuft"	T 175	TIMER	// Safety-Integrated Hardwaretest läuft verlängert (1 sek.)
"Ta_M_Reset_Taste"	T 176	TIMER	// Reset Taste verlängert (2 sek.)
"Te_WIKO_Main"	T 177	TIMER	// Timer für Baustein FC_WIKO_MAIN
"Ta_WZW_Aktiv"	T 178	TIMER
"Te_G0_Timer_Fehler"	T 179	TIMER
"T_SOKO"	T 180	TIMER
"T_Laufzeit_Vlies"	T 181	TIMER
"T_KSA3_Entpr_Vlies_EIN"	T 182	TIMER
"TE_Prg_nicht_aktiv"	T 183	TIMER	// Verzögerung Programm läuft nicht
"Te_Pnoz_Freigabe"	T 184	TIMER	// Verzögerung des Fehlers bei fehlender Pnoz-Freigabe
"Te_Klemm_Ueb"	T 185	TIMER
"T_KSA7_SPALTSIEB_LAUFZ"	T 186	TIMER	// KSA7: Laufzeitüberwachung Spaltsieb-Zylinder
"Ta_LS_Auftrag_laeuft"	T 187	TIMER
"TV_M30_Reset"	T 188	TIMER	// Verlängerter Impuls M30 oder Taste Reset
"Ta_Verz_Abfr_Trans"	T 189	TIMER
"T_KSA3_KSA7_MAX"	T 190	TIMER	// KSA3_KSA7: Verzögerung Füllstand maximum
"T_KSA3_KSA7_MIN"	T 191	TIMER	// KSA3_KSA7: Verzögerung Füllstand minimum
"T_KSA3_KSA7_VORW"	T 192	TIMER	// KSA3_KSA7: Verzögerung Füllstand Vorwarnung
"T_KSA3_KSA7_VORW_REAKT"	T 193	TIMER
"T_KSA3_Vlies_max_Lau"	T 194	TIMER
"Te_GetriebeS_undefiniert"	T 195	TIMER
"T_wgfTWa"	T 196	TIMER	// Wzw.Grundstellung fahren Schritt Wartezeit
"T_vwgfTUe"	T 197	TIMER	// vert. Wzw.Grundstellung fahren Schritt Überwachungszeit
"Ta_Vorbereiten_aktiv"	T 198	TIMER	// Reserve
"T_Messd_abbl"	T 199	TIMER	// Timer Blasluft Reinigung Werkzeugvermessung |
"Tv_Soko1"	T 200	TIMER
"T_SPI_Schmierung1"	T 201	TIMER
"T_SPI_Schmierung2"	T 202	TIMER
"T_SPI_Schmierung3"	T 203	TIMER
"T_SPI_Schmierung4"	T 204	TIMER
"T_SPI_Schmierung5"	T 205	TIMER
"Te_Kein_WZ_IN_SPI"	T 206	TIMER	// Te für "Kein Werkzeug in Spindel"
"Te_SpH_MPL_FG_verz"	T 207	TIMER	// TE: Freigabe Spannhydraulik im MPL verzögert
"SE_HAWE_Lebenszeichen"	T 208	TIMER	// HAWE-Lebenszeichen vom ProfiBus
"SA_PW_Rettungsbilder"	T 209	TIMER	// Rettungsbild PW1/PW2/PW3 ist angewählt
"T_KSA3.1_Meldung"	T 210	TIMER	// Timer für Baustein KSA3.1 für Funktion Meldung
"T_KSA3.1_Reaktion"	T 211	TIMER	// Timer für KSA3.1 Funktion: Reaktion
"T_KSA3.1_Kratz"	T 212	TIMER	// Timer für KSA3.1 Funktion:Kratzbandförderer
"Te_Ueb_Pin_Lock"	T 213	TIMER
"Te_Ueb_Pin_Mag_Lock"	T 214	TIMER
"Te_Pin_Ruest_Lock"	T 215	TIMER
"Ta_wgfStrt"	T 216	TIMER	// sa Wzw.Grundstellung fahren Start
"Tv_T_KabTuer_entriegeln"	T 217	TIMER	// Verlängerter Impuls Taste Kabinentür entriegeln
"Tv_OEM_Maskenumschaltung"	T 218	TIMER	// Zeitverzögerung für Maskenumschaltung OEM-Rettung
"Ta_Mag_manuell"	T 219	TIMER	// Abfallverzögerung Magazin drehen Hand
"Te_FD_Tisch_Temp2"	T 220	TIMER
"Te_FD_Tisch_Temp1"	T 221	TIMER
"Te_SP_RPL_Gespannt"	T 222	TIMER	// Verzögerter Impuls für Spannhydraulik am Rüstplatz gespannt
"Te_SPH_SCH_Schmierimpuls"	T 223	TIMER	// Verzögerter Impuls für maximale Schmierdauer
"Te_SPH_SCH_Druck_nicht_0"	T 224	TIMER	// Verzögerter Impuls SPH Schmierung Druck nicht 0
"Te_SPH_SCH_Druck_ok"	T 225	TIMER	// Verzögerter Impuls SPH Schmierung Druck ok
"SV_RPL_abblasen"	T 226	TIMER	// Zeitimpuls Vorrichtung am Rüstplatz abblasen Stelle 1+2
"Te_AUTO_TPU_TRANSFERPOS"	T 227	TIMER
"Te_SPH_MPL_RPL_Filter"	T 228	TIMER	// Einschaltverzögerung Spannhydraulik Filter verschmutzt
"Te_Achs15"	T 229	TIMER	// Timer Einschaltverzögert AX 15-Achse: Bremse lösen
"Te_Getriebeschaltung"	T 230	TIMER	// Verzögerung Getriebe geschaltet
"Te_PW_GRST_verz"	T 231	TIMER	// PW-Ablauf in Grundstellung verzögert
"T_PwgTWa"	T 232	TIMER	// PalWechsel Grundstellung fahren Schritt Wartezeit
"T_PwgTUe"	T 233	TIMER	// PalWechsel Grundstellung fahren Schritt Überwachungszeit
"T_PRG_LAEUFT_VERZ"	T 234	TIMER	// Programm läuft in Automatik verzögert
"Ta_PwgSt"	T 235	TIMER	// sa PalWechsel Grundstellung fahren SrKette Start
"T_SAFECO_Pnotz_0_setzten"	T 236	TIMER
"T_SAFECO_ZD_Schritt[3]"	T 237	TIMER
"Tv_Absau_Time"	T 238	TIMER	// Timer erhoeht Absaugung
"Ta_TPU_UEB_ENTPR"	T 239	TIMER
"T_SAFECO_Maschine_Ein"	T 240	TIMER	// Verzögerung Maschine Ein
"T_SAFECO_Override_100"	T 241	TIMER	// Override 3 sec auf 100 %
"T_SAFECO_ZD_Override100"	T 242	TIMER
"T_SAFECO_GR1ZD_Schritt_2"	T 243	TIMER	// ZD Bereich 1 Bremsen in hängenden Achsen (3+5) eingefallen verzögert
"T_SAFECO_Bremsentest_1"	T 244	TIMER	// Bremsentest 1 ( vertikale Achse )
"T_SAFECO_Bremsentest_2"	T 245	TIMER	// Bremsentest 2 ( Kopf - Achse )
"T_SAFECO_STOPA_SPI"	T 246	TIMER	// Verzögerung StopC StopA Spindel
"T_NH_STOPA_AX"	T 247	TIMER	// Ausschaltverzögerung  SPL M_NOT_HALT_AX
"Te_SpiKlemm_beide_0Signa"	T 248	TIMER	// Eingänge Klemmung Spindel beide 0-Signal verzögert
"T_SAFECO_Bremsentest_3"	T 249	TIMER	// Bremsentest 3 ( Palettenspeicher Hub - Achse )
"T_SAFECO_GR2ZD_Schritt_2"	T 250	TIMER	// Bereich 2 ZD Bremsen in hängenden Achsen (16) eingefallen verzögert
"T_SA_GR2ZD_HWTest_laeuft"	T 251	TIMER	// Bereich 2 PS Safety-Integrated Hardwaretest läuft verlängert (1 sek.)
"T_SAFECO_SST_DRIV_EN_CNC"	T 252	TIMER	// Antriebsfreigabe von PNOZ für Rüstplatzachse abfallverzögert
"T_SAFECO_Err_BA3"	T 253	TIMER	// Überwachungszeit BA 1
"T_SAFECO_Err_BA4"	T 254	TIMER	// Überwachungszeit BA 1
"Te_HAWE_Lebenszeichen"	T 255	TIMER	// Überwachung HAWE-Lebenszeichen
"Te_SpH_Aggregat_ein"	T 256	TIMER	// Meldung: SpannHydraulik Aggregat ist ein
"Te_MPL_Kupplung"	T 257	TIMER	// Überwachung MPL Kupplung Spannhydraulik
"Te_Pin_Ruest_Unlock"	T 259	TIMER
"Te_Z_Achse_inPos"	T 260	TIMER	// Verzögerung Z-Achse in Position
"Tv_MCU_Prg_Start"	T 261	TIMER	// 100ms-Impuls für MCU Programm-Anfang
"Te_MCU_Grenzen_RESET"	T 262	TIMER	// MCU: RESET Grenzen aktivieren / deaktivieren
"Tv_WMT_zu"	T 263	TIMER	// Impuls WZ-Magazin-Tür wurde geschlossen
"Te_REF_SPI_Error"	T 264	TIMER	// Einschaltverzögerung Spindel Referenzlauf fehlgeschlagen
"Te_RPL_Feh_Tuer"	T 265	TIMER	//  Ruestplatz  Fehlbedienung RPL-Tuer nicht offen
"Te_Konen_ausblasen"	T 266	TIMER	// Timer Konen ausblasen
"Te_Schalterk_MPL_anw"	T 267	TIMER	// Timer MPL Schalterkontrolle
"Tv_PW_Time_spuel_senk"	T 268	TIMER	// Timer Spuelzeit PW-Hub senken ohne Positionsschalter4
"Tv_Messtaster_Fehler2"	T 269	TIMER
"T_SPDL_Komp"	T 270	TIMER	// Timer für Glättungskompensation GMN Spindel
"Tv_Kalibrierring_ablasen"	T 271	TIMER	// Abblaszeit für Kalibrierring
"te_Roboter_LZ_0_Signal"	T 272	TIMER	// Datenüberwachung Roboter Laufzeit 0-Signal
"te_Roboter_LZ_1_Signal"	T 273	TIMER	// Datenüberwachung Roboter Laufzeit 1-Signal
"Te_Max_RPL_Dusche"	T 274	TIMER	// max. Laufzeit Rüstplatz-Dusche in [10s]
"Te_Ma_Pl_belegt"	T 275	TIMER	// Timer: Signal Palette vorhanden
"Ta_Rett_Time"	T 276	TIMER	// verzoegerte Rettungssignale
"T_Verz_WZ_entl_meld"	T 279	TIMER
"TE_SF_FRG_Tuer"	T 280	TIMER	// Freigabe Timer  Tuer oeffnen
"T_Ueberw_Drucklos"	T 281	TIMER	// Ueberwachung  Drucklos
"T_SF_FP2_Zur_R1"	T 282	TIMER	// Rechen 1 vor/zurueck
"T_SF_FP2_Zur_R2"	T 283	TIMER	// Rechen 2 vor/zurück
"Te_Greifer_in_Bewegung"	T 284	TIMER	// Greifer aus- einfahren aktiv verzögert
"Te_MPL_vers_2_Hubb"	T 285	TIMER	// 2.Hubbeweung wenn die Schalterkontrolle keinen korrekten Zustand meldet
"Te_Achs19"	T 286	TIMER
"Te_Achs18"	T 287	TIMER
"Te_Ruest_Verr2_Verz"	T 289	TIMER
"Tv_Maschine_ein_aus"	T 290	TIMER	// Maschine Ein / Aus verlängerter Impuls
"Te_RPL_Druck_0"	T 291	TIMER	// FD: Rüstplatz Druck_0 verzögert an HAWE
"Tv_WZ_Datensicherung"	T 292	TIMER	// Anstoss Datensicherung Werkzeugdaten
"Te_Start_ReadAccessLevel"	T 293	TIMER	// Zeitverzögertes Starten für AccessLevel lesen
"Tv_Smartkey_Ident_Senden"	T 294	TIMER	// Signal von angelegten Tag mindestens 500ms senden
"TE_IKZ_OVERRIDE_0"	T 296	TIMER	// KM: Override 0 durch innere Kühlmittelzufuhr aktiv
"Tvi_LZ_Kegelreinigung"	T 297	TIMER	// Verlängerter Impuls Kegelreinigung
"T_KSA7_DS_UNTERDRUCK"	T 298	TIMER	// KSA7: Druckschalter Unterdruck IKZ entprellt
"T_KNOLL_verz"	T 299	TIMER
"t_pw_schmier_fuellstand"	T 300	TIMER	// Palettenwechsler: Schmierung Füllstand unterschritten verzögert
"t_pw_schmier_eing_verz"	T 301	TIMER	// Palettenwechsler: Schmierung eingeschaltet verzögert
"t_pw_schmier_ausg_verz"	T 302	TIMER	// Palettenwechsler: Schmierung ausgeschaltet verzögert
"T_WZW_HEBEPUMPE_EIN"	T 303	TIMER	// Werkzeugwechsler: Hebepumpe einschalten verlängerter Impuls
"Te_Achs16"	T 304	TIMER	// Timer Einschaltverzögert AX 16-Achse: Bremse lösen
"Te_ALK_entlueften"	T 305	TIMER	// Timer Laufzeit Auflagenkontrolle "Luft-Reinigung" entlüften
"Te_SPH_Druck0_fehlt"	T 306	TIMER	// Timer Spannhydraulik Druck=0 fehlt
"TE_Mag_Verr2_Verz"	T 309	TIMER
"T_Bremsen_Zu_verz_ESR"	T 310	TIMER	// DM_ESR: Verzögertes abschalten der Bremsen um Rückzug zu gewährleisten
"Te_PW_MPL_belegt"	T 311	TIMER	// Einschaltverzögerung: Entprellen von IX_PW_MPL_belegt
"Te_PW_PNOZ_FG"	T 314	TIMER	// PW-PNOZ-Freigabe verzögert für "Leistung aktiv Achse 8"
"Te_WM_Energiefreigabe"	T 315	TIMER	// FM 701138 "SPI-VS-H, 7.Achse nicht bereit (Drive ready fehlt) um 500ms verzögert
"te_FM_700350"	T 319	TIMER	// Einschaltverzögerung der Fehlermeldung Magazinklappe nicht geschlossen
"Te_Smartkey_ErrorReset"	T 320	TIMER
"T_Verzög_Reset"	T 321	TIMER
"T_KSA3_KSA_Mel_Entprelle"	T 329	TIMER
"T_SE_TAKT_POS"	T 330	TIMER	// Dauer Positiver Zustand des Takt
"T_SE_TAKT_NEG"	T 331	TIMER	// Dauer Negativer Zustand des Takt
"T_SE_Roboter_Sync"	T 332	TIMER
"T_SE_Robot_Verzug"	T 333	TIMER
"T_SE_WERKSTUECK_W_OK"	T 334	TIMER	// Zeit für Roboter Werkstückwechsel o.k.
"T_SE_BELADEN_ENDE"	T 335	TIMER	// min. 200msec muss Beladenende anstehen um gültig zu sein
"Tv_RPL_NachCTRL_unterdr"	T 336	TIMER	// TV: Rüstplatz Nachregeln unterdrücken (NOTAUS von Hawe steht an)
"Tv_FD_FM_Regelung"	T 337	TIMER	// FD-Spannhydraulik: FM "Druck beim Regeln nicht erreichbar" verzögert auswerten
"T_SV_Startimpuls_MSST"	T 340	TIMER
"Te_Pos_Brush_clean"	T 350	TIMER
"Ta_WZW_Aktiv_beendet"	T 351	TIMER
"TE_REQ_DRV_1_READY"	T 370	TIMER	// Verzögerte Abfrage des Nahtstellensignals DRIVE  READY Achse 1 (DBX93.5)
"TE_REQ_DRV_2_READY"	T 371	TIMER	// Verzögerte Abfrage des Nahtstellensignals DRIVE  READY Achse 2 (DBX93.5)
"TE_REQ_DRV_3_READY"	T 372	TIMER	// Verzögerte Abfrage des Nahtstellensignals DRIVE  READY Achse 3 (DBX93.5)
"TE_REQ_DRV_4_READY"	T 373	TIMER	// Verzögerte Abfrage des Nahtstellensignals DRIVE  READY Achse 4 (DBX93.5)
"TE_REQ_DRV_5_READY"	T 374	TIMER	// Verzögerte Abfrage des Nahtstellensignals DRIVE  READY Achse 5 (DBX93.5)
"TE_REQ_DRV_6_READY"	T 375	TIMER	// Verzögerte Abfrage des Nahtstellensignals DRIVE  READY Achse 6 (DBX93.5)
"TE_REQ_DRV_7_READY"	T 376	TIMER	// Verzögerte Abfrage des Nahtstellensignals DRIVE  READY Achse 7 (DBX93.5)
"TE_REQ_DRV_8_READY"	T 377	TIMER	// Verzögerte Abfrage des Nahtstellensignals DRIVE  READY Achse 8 (DBX93.5)
"TE_REQ_DRV_9_READY"	T 378	TIMER	// Verzögerte Abfrage des Nahtstellensignals DRIVE  READY Achse 9 (DBX93.5)
"TE_REQ_DRV_10_READY"	T 379	TIMER	// Verzögerte Abfrage des Nahtstellensignals DRIVE  READY Achse 10 (DBX93.5)
"TE_REQ_DRV_11_READY"	T 380	TIMER	// Verzögerte Abfrage des Nahtstellensignals DRIVE  READY Achse 11 (DBX93.5)
"TE_REQ_DRV_12_READY"	T 381	TIMER	// Verzögerte Abfrage des Nahtstellensignals DRIVE  READY Achse 12 (DBX93.5)
"TE_REQ_DRV_13_READY"	T 382	TIMER	// Verzögerte Abfrage des Nahtstellensignals DRIVE  READY Achse 13 (DBX93.5)
"TE_REQ_DRV_14_READY"	T 383	TIMER	// Verzögerte Abfrage des Nahtstellensignals DRIVE  READY Achse 14 (DBX93.5)
"TE_REQ_DRV_15_READY"	T 384	TIMER	// Verzögerte Abfrage des Nahtstellensignals DRIVE  READY Achse 15 (DBX93.5)
"TE_REQ_DRV_16_READY"	T 385	TIMER	// Verzögerte Abfrage des Nahtstellensignals DRIVE  READY Achse 16 (DBX93.5)
"TE_REQ_DRV_17_READY"	T 386	TIMER	// Verzögerte Abfrage des Nahtstellensignals DRIVE  READY Achse 17 (DBX93.5)
"TE_REQ_DRV_18_READY"	T 387	TIMER	// Verzögerte Abfrage des Nahtstellensignals DRIVE  READY Achse 18 (DBX93.5)
"TE_REQ_DRV_19_READY"	T 388	TIMER	// Verzögerte Abfrage des Nahtstellensignals DRIVE  READY Achse 19 (DBX93.5)
"TE_REQ_DRV_20_READY"	T 389	TIMER	// Verzögerte Abfrage des Nahtstellensignals DRIVE  READY Achse 20 (DBX93.5)
"T_E_MAPAL_Enable_Axis"	T 400	TIMER	// Verzögerte Reglerfreigabe U-Achse Mapal
"T_E_MAPAL_Disable_Axis"	T 401	TIMER	// Verzögerte Reglersperre U-Achse Mapal
"T_VI_MAPAL_Quit_Error"	T 402	TIMER	// Impuls für Fehlerquittierung U-Achse Mapal
"T_E_MAPAL_ERR_not_ready"	T 403	TIMER	// Verzögerung für Fehler U-Achse Mapal not ready
"T_E_MAPAL_QUIT_M144"	T 404	TIMER	// Verzögerte Quittierung der M-Funktion M144 U-Achse Mapal
"T_E_MAPAL_QUIT_H68"	T 405	TIMER	// Verzögerte Quittierung der H-Funktion H68 U-Achse Mapal
"Te_Clock_Time"	T 450	TIMER
"Te_Entpr_LA_Klappe"	T 451	TIMER	// Fehlererkennung externe Eingänge
"TE_PW_AKTIV_VERZ"	T 497	TIMER	// Palettenwechsler aktiv verzögert
"TE_MSS_KUEHLUNG_VERZ"	T 498	TIMER	// Motorschutzschalter Schaltschrankkühlung hat ausgelöst verzögert
"T_TAKTTISCH_IN_POS_VERZ"	T 499	TIMER	// Takttisch in Position verzögert
"t_technische_stoerung"	T 500	TIMER	// HMI-PRO: Technische Störung verzögert
"t_taktzeitmessung"	T 501	TIMER	// HMI-PRO: Zeitstufe für Taktzeitmesung
"TE_ENABLE_OUT_3_NX_NCU"	T 507	TIMER	// Klemme X122.2 AUS3 verz. (Leistung eingeschaltet)
"TE_NCU_KL122_1_SLM_BTB"	T 508	TIMER	// Ansteuerung NCU: Klemme X122.1 SLM bereit verz.
"TE_NCU_KL122_2_AUS3"	T 509	TIMER	// Ansteuerung NCU: Abschalten der Klemme X122.2 AUS3 verz.
"TE_MASCHINE_AUS"	T 510	TIMER	// Maschine Aus verzögert
"TE_MASCHINE_EIN"	T 511	TIMER	// Maschine Ein verzögert
"UDT_DB2_PLC_MESSAGE"	UDT 2	UDT 2	// UDT für DB 2 Interface for Alarms & Messages
"UDT_DB10_SIEM_NCK"	UDT 10	UDT 10	// UDT für DB 10 Interface NCK
"UDT_DB11_SIEM_BAG"	UDT 11	UDT 11	// UDT für DB 11 Interface BAG
"UDT_DB19_SIEM_MMC"	UDT 19	UDT 19	// UDT für DB 19 Interface MMC-Signals
"UDT_PLC_MD_DB20"	UDT 20	UDT 20	// UDT für DB 20 Maschinen-Konfiguration
"UDT_DB21_SIEM_KANAL1"	UDT 21	UDT 21	// UDT für DB 21 Interface Chanel 1
"UDT_DBS_ACHSEN"	UDT 31	UDT 31	// UDT für Interface Achsen
"UDT_TRANSLINE"	UDT 59	UDT 59	// UDT für DB 59 Schnittstelle zu HMI PRO
"UDT_62"	UDT 62	UDT 62
"UDT_65"	UDT 65	UDT 65	// UDT für DB65 Datenbaustein Familienmodul
"UDT_NC_PLC_DB70"	UDT 70	UDT 70	// UDT für DB 70 DUAL-Port-RAM: Datentausch NC<==>PLC
"UDT_DB71_TMLoadIF"	UDT 71	UDT 71	// UDT für DB70 Interface loading-/unloadingstation for Toolmanagment
"UDT_DB72_TMSpindleIF"	UDT 72	UDT 72	// UDT für DB72 Interface Spindle for Toolmanagment
"UDT_DB73_Revolver"	UDT 73	UDT 73	// UDT für DB73 Interface Revolver for Toolmanagment
"UDT_DP_DIAG"	UDT 78	UDT 78	// DP-Diagnose für Sinumerik-Wizard
"UDT100"	UDT 100	UDT 100	// UDT für DB100 "DB_Remanent"
"UDT_HMI_PRO_ADD"	UDT 159	UDT 159	// UDT für DB 159 Schnittstelle zu HMI PRO Erweiterung
"UDT_VWWZ"	UDT 175	UDT 175	// UDT für DB175: vert.Werkzeugwechsler Grdstlg.fahren...
"UDT_WWZ"	UDT 176	UDT 176	// UDT für DB176: WzVerwaltung Grdstlg.fahren...
"UDT_ASUP_MACHINE"	UDT 201	UDT 201	// UDT für DB201 ASUP Maschine
"UDT_Datenpunkt_TDS"	UDT 228	UDT 228	// UDT für DB228: TDS
"UDT_DB240_MSG_AEND"	UDT 240	UDT 240	// UDT für DB240: DB_MSG_AEND   Fehlereintrag an SOKO
"UDT_ALG"	UDT 254	UDT 254	// allgemeine Signale
"UDT_NC_PLC_Zusatz"	UDT 701	UDT 701
"UDT_VWWZ_0"	UDT 1751	UDT 1751	// zu UDT_WWZ und stat.Daten FC_WZW_VMAG_STATUS
"UDT_WWZ_0"	UDT 1761	UDT 1761	// zu UDT_VWWZ und stat.Daten FC_WZW_STATUS
"V_Omron"	VAT 3	
"HAWE"	VAT 4	
"Fehler_WZW"	VAT 5	
"VATm-fkt"	VAT 6	
"M_FKT_Test"	VAT 7	
"VAT_WZV_Fehler"	VAT 8	
"safe"	VAT 9	
"VATvibs"	VAT 10	
"VATvibs(1)"	VAT 11	
"VAT_Icons"	VAT 12	
"zd"	VAT 13	
"VatOEM"	VAT 14	
"VAT_RS"	VAT 15	
"VAT_RS1"	VAT 16	
"VAT_tempcomp"	VAT 17	
"TDS_db137_geisl"	VAT 18	
"TDS_2"	VAT 19	
"TDS_3"	VAT 20	
"TDS_4"	VAT 21	
"Sintdi"	VAT 22	
"V_DB71"	VAT 23	
"TDS_WDVT"	VAT 24	
"V_SOKO_ERROR"	VAT 25	
"VAT_SPH_Systemparameter"	VAT 26		// UDT_INT-Parameter
"VAT_Rob_BoschRexroth_MPL"	VAT 27	
"VAT_SPH_MA_St1"	VAT 28	
"VAT_SPH_RP_St2"	VAT 29	
"BL_MESST"	VAT 33	
"VAT_SpH_Teachen"	VAT 34	
"VAT_SPH_RP_St1"	VAT 35	
"VAT_CTS"	VAT 36	
"VAT_KMTL_KNOLL"	VAT 37	
"VAT_Schritte_Teller"	VAT 38	
"SI"	VAT 39	
"V_KometUAx"	VAT 40	
"VAT_SPH_RP_St1_RS"	VAT 43	
"TDS_db137"	VAT 44	
"TDS_db227"	VAT 45	
"VAT_Rob_BoschRexroth:RPL"	VAT 46	
"VAT_Wiegekopf"	VAT 47	
"VAT_HAWEtest"	VAT 49	
"TDS_baltic"	VAT 50	
"VAT_UMKS_KETTE"	VAT 51	
"VAT_PW_heb_senk"	VAT 52	
"VAT_PW_handrad"	VAT 53	
"V_WwGf"	VAT 55		// Test Wzw.Grundstlg.fahren
"VAT_MSST"	VAT 56	
"VAT_BAG"	VAT 57	
"MCP"	VAT 58	
"VAT_Achs_DB36"	VAT 59	
"VAT_60"	VAT 60		// Eingänge
"TESTSTOP_VAT"	VAT 61	
"VAT_wzw"	VAT 62	
"VAT_RS10"	VAT 63	
"VAT_HGC2"	VAT 64	
"VAT_Roboter"	VAT 65	
"VAT_HGC"	VAT 66	
"VAT_AutoRPL_Tuer"	VAT 67	
"VAT_Roboter_Allg"	VAT 68	
"VAT_Rob_Sonder"	VAT 69	
"VAT_ws"	VAT 70	
"VAT_71"	VAT 71	
END_SYMBOL_TABLE
